LIN {X 0.039,Y -394.828,Z 1620.610,A 0.000,B 0.000,C 90.000,E1 109.812} C_DIS
LIN {X -0.087,Y -410.950,Z 1620.598,A 0.000,B 0.000,C 90.000,E1 107.583} C_DIS
LIN {X 0.069,Y -428.624,Z 1620.585,A 0.000,B 0.000,C 90.000,E1 105.371} C_DIS
LIN {X 0.081,Y -447.896,Z 1620.574,A 0.000,B 0.000,C 90.000,E1 103.244} C_DIS
LIN {X -0.189,Y -468.016,Z 1620.563,A 0.000,B 0.000,C 90.000,E1 101.299} C_DIS
LIN {X -0.227,Y -491.296,Z 1620.551,A 0.000,B 0.000,C 90.000,E1 99.265} C_DIS
LIN {X 0.069,Y -496.545,Z 1620.549,A 0.000,B 0.000,C 90.000,E1 98.803} C_DIS
LIN {X -0.222,Y -498.760,Z 1620.548,A 0.000,B 0.000,C 90.000,E1 98.624} C_DIS
LIN {X -0.096,Y -500.441,Z 1620.547,A 0.000,B 0.000,C 90.000,E1 98.398} C_DIS
LIN {X -0.170,Y -501.913,Z 1620.545,A 0.000,B 0.000,C 90.000,E1 98.163} C_DIS
LIN {X 0.252,Y -503.003,Z 1620.544,A 0.000,B 0.000,C 90.000,E1 97.871} C_DIS
LIN {X 0.048,Y -504.268,Z 1620.541,A 0.000,B 0.000,C 90.000,E1 97.409} C_DIS
LIN {X -0.150,Y -504.485,Z 1620.538,A 0.000,B 0.000,C 90.000,E1 96.947} C_DIS
LIN {X 0.160,Y -503.694,Z 1620.536,A 0.000,B 0.000,C 90.000,E1 96.429} C_DIS
LIN {X -0.030,Y -501.759,Z 1620.533,A 0.000,B 0.000,C 90.000,E1 95.967} C_DIS
LIN {X 0.225,Y -498.522,Z 1620.530,A 0.000,B 0.000,C 90.000,E1 95.454} C_DIS
LIN {X 0.209,Y -485.108,Z 1620.520,A 0.000,B 0.000,C 90.000,E1 93.498} C_DIS
LIN {X 0.202,Y -474.979,Z 1620.511,A 0.000,B 0.000,C 90.000,E1 92.007} C_DIS
LIN {X 0.024,Y -464.430,Z 1620.503,A 0.000,B 0.000,C 90.000,E1 90.516} C_DIS
LIN {X 0.121,Y -453.568,Z 1620.494,A 0.000,B 0.000,C 90.000,E1 88.969} C_DIS
LIN {X -0.158,Y -444.053,Z 1620.487,A 0.000,B 0.000,C 90.000,E1 87.707} C_DIS
LIN {X 0.033,Y -432.154,Z 1620.478,A 0.000,B 0.000,C 90.000,E1 86.102} C_DIS
LIN {X -0.096,Y -416.231,Z 1620.466,A 0.000,B 0.000,C 90.000,E1 83.970} C_DIS
LIN {X -0.079,Y -399.065,Z 1620.453,A 0.000,B 0.000,C 90.000,E1 81.489} C_DIS
LIN {X 0.091,Y -381.295,Z 1620.437,A 0.000,B 0.000,C 90.000,E1 78.634} C_DIS
LIN {X -0.092,Y -366.244,Z 1620.422,A 0.000,B 0.000,C 90.000,E1 76.047} C_DIS
LIN {X -0.121,Y -354.890,Z 1620.411,A 0.000,B 0.000,C 90.000,E1 73.976} C_DIS
LIN {X 0.056,Y -339.308,Z 1620.394,A 0.000,B 0.000,C 90.000,E1 70.913} C_DIS
LIN {X 0.117,Y -325.813,Z 1620.378,A 0.000,B 0.000,C 90.000,E1 68.103} C_DIS
LIN {X 0.153,Y -310.778,Z 1620.359,A 0.000,B 0.000,C 90.000,E1 64.588} C_DIS
LIN {X -0.117,Y -301.768,Z 1620.346,A 0.000,B 0.000,C 90.000,E1 62.359} C_DIS
LIN {X 0.106,Y -292.615,Z 1620.333,A 0.000,B 0.000,C 90.000,E1 59.999} C_DIS
LIN {X 0.041,Y -284.397,Z 1620.322,A 0.000,B 0.000,C 90.000,E1 57.995} C_DIS
LIN {X 0.019,Y -277.272,Z 1620.313,A 0.000,B 0.000,C 90.000,E1 56.294} C_DIS
LIN {X 0.123,Y -268.440,Z 1620.301,A 0.000,B 0.000,C 90.000,E1 54.196} C_DIS
LIN {X 0.060,Y -258.267,Z 1620.287,A 0.000,B 0.000,C 90.000,E1 51.743} C_DIS
LIN {X 0.110,Y -247.009,Z 1620.271,A 0.000,B 0.000,C 90.000,E1 48.852} C_DIS
LIN {X -0.019,Y -235.570,Z 1620.253,A 0.000,B 0.000,C 90.000,E1 45.567} C_DIS
LIN {X 0.043,Y -225.173,Z 1620.234,A 0.000,B 0.000,C 90.000,E1 42.162} C_DIS
LIN {X -0.046,Y -216.778,Z 1620.217,A 0.000,B 0.000,C 90.000,E1 39.116} C_DIS
LIN {X -0.102,Y -209.208,Z 1620.200,A 0.000,B 0.000,C 90.000,E1 36.011} C_DIS
LIN {X -0.074,Y -202.410,Z 1620.182,A 0.000,B 0.000,C 90.000,E1 32.832} C_DIS
LIN {X 0.013,Y -196.332,Z 1620.164,A 0.000,B 0.000,C 90.000,E1 29.589} C_DIS
LIN {X -0.096,Y -190.985,Z 1620.146,A 0.000,B 0.000,C 90.000,E1 26.360} C_DIS
LIN {X 0.019,Y -186.372,Z 1620.128,A 0.000,B 0.000,C 90.000,E1 23.025} C_DIS
LIN {X 0.023,Y -181.503,Z 1620.105,A 0.000,B 0.000,C 90.000,E1 18.852} C_DIS
LIN {X -0.016,Y -177.501,Z 1620.081,A 0.000,B 0.000,C 90.000,E1 14.647} C_DIS
LIN {X 0.063,Y -174.184,Z 1620.058,A 0.000,B 0.000,C 90.000,E1 10.366} C_DIS
LIN {X 0.061,Y -171.420,Z 1620.029,A 0.000,B 0.000,C 90.000,E1 5.220} C_DIS
LIN {X 0.000,Y -169.706,Z 1620.000,A 0.000,B 0.000,C 90.000,E1 360.000} C_DIS
LIN {X 0.005,Y -170.849,Z 1619.930,A 0.000,B 0.000,C 90.000,E1 347.409} C_DIS
LIN {X 0.018,Y -173.863,Z 1619.901,A 0.000,B 0.000,C 90.000,E1 342.236} C_DIS
LIN {X -0.034,Y -177.684,Z 1619.878,A 0.000,B 0.000,C 90.000,E1 337.975} C_DIS
LIN {X -0.054,Y -181.799,Z 1619.859,A 0.000,B 0.000,C 90.000,E1 334.588} C_DIS
LIN {X 0.104,Y -186.773,Z 1619.840,A 0.000,B 0.000,C 90.000,E1 331.179} C_DIS
LIN {X 0.076,Y -192.581,Z 1619.822,A 0.000,B 0.000,C 90.000,E1 327.867} C_DIS
LIN {X 0.010,Y -199.125,Z 1619.803,A 0.000,B 0.000,C 90.000,E1 324.609} C_DIS
LIN {X 0.022,Y -206.480,Z 1619.785,A 0.000,B 0.000,C 90.000,E1 321.376} C_DIS
LIN {X -0.028,Y -213.691,Z 1619.770,A 0.000,B 0.000,C 90.000,E1 318.609} C_DIS
LIN {X -0.020,Y -222.947,Z 1619.753,A 0.000,B 0.000,C 90.000,E1 315.486} C_DIS
LIN {X -0.099,Y -233.261,Z 1619.736,A 0.000,B 0.000,C 90.000,E1 312.447} C_DIS
LIN {X 0.021,Y -240.378,Z 1619.725,A 0.000,B 0.000,C 90.000,E1 310.539} C_DIS
LIN {X -0.047,Y -248.275,Z 1619.715,A 0.000,B 0.000,C 90.000,E1 308.705} C_DIS
LIN {X 0.038,Y -258.830,Z 1619.703,A 0.000,B 0.000,C 90.000,E1 306.503} C_DIS
LIN {X 0.074,Y -274.871,Z 1619.687,A 0.000,B 0.000,C 90.000,E1 303.658} C_DIS
LIN {X 0.052,Y -288.392,Z 1619.676,A 0.000,B 0.000,C 90.000,E1 301.592} C_DIS
LIN {X -0.139,Y -307.952,Z 1619.661,A 0.000,B 0.000,C 90.000,E1 298.949} C_DIS
LIN {X -0.148,Y -322.812,Z 1619.650,A 0.000,B 0.000,C 90.000,E1 297.001} C_DIS
LIN {X -0.137,Y -335.094,Z 1619.641,A 0.000,B 0.000,C 90.000,E1 295.412} C_DIS
LIN {X 0.086,Y -349.411,Z 1619.631,A 0.000,B 0.000,C 90.000,E1 293.515} C_DIS
LIN {X -0.020,Y -363.824,Z 1619.621,A 0.000,B 0.000,C 90.000,E1 291.716} C_DIS
LIN {X -0.061,Y -373.411,Z 1619.614,A 0.000,B 0.000,C 90.000,E1 290.536} C_DIS
LIN {X 0.121,Y -380.238,Z 1619.609,A 0.000,B 0.000,C 90.000,E1 289.631} C_DIS
LIN {X 0.023,Y -388.598,Z 1619.603,A 0.000,B 0.000,C 90.000,E1 288.489} C_DIS
LIN {X -0.017,Y -394.281,Z 1619.598,A 0.000,B 0.000,C 90.000,E1 287.638} C_DIS
LIN {X -0.182,Y -397.729,Z 1619.595,A 0.000,B 0.000,C 90.000,E1 287.094} C_DIS
LIN {X 0.129,Y -402.189,Z 1619.590,A 0.000,B 0.000,C 90.000,E1 286.205} C_DIS
LIN {X 0.097,Y -405.842,Z 1619.585,A 0.000,B 0.000,C 90.000,E1 285.371} C_DIS
LIN {X -0.002,Y -407.799,Z 1619.582,A 0.000,B 0.000,C 90.000,E1 284.828} C_DIS
LIN {X -0.201,Y -409.417,Z 1619.579,A 0.000,B 0.000,C 90.000,E1 284.300} C_DIS
LIN {X 0.013,Y -410.583,Z 1619.576,A 0.000,B 0.000,C 90.000,E1 283.716} C_DIS
LIN {X -0.066,Y -411.312,Z 1619.573,A 0.000,B 0.000,C 90.000,E1 283.175} C_DIS
LIN {X 0.166,Y -411.580,Z 1619.570,A 0.000,B 0.000,C 90.000,E1 282.591} C_DIS
LIN {X 0.003,Y -411.346,Z 1619.567,A 0.000,B 0.000,C 90.000,E1 282.063} C_DIS
LIN {X -0.160,Y -410.620,Z 1619.564,A 0.000,B 0.000,C 90.000,E1 281.535} C_DIS
LIN {X 0.078,Y -409.270,Z 1619.561,A 0.000,B 0.000,C 90.000,E1 280.950} C_DIS
LIN {X -0.092,Y -407.390,Z 1619.558,A 0.000,B 0.000,C 90.000,E1 280.423} C_DIS
LIN {X 0.059,Y -404.789,Z 1619.555,A 0.000,B 0.000,C 90.000,E1 279.849} C_DIS
LIN {X -0.136,Y -401.553,Z 1619.552,A 0.000,B 0.000,C 90.000,E1 279.321} C_DIS
LIN {X -0.015,Y -397.674,Z 1619.549,A 0.000,B 0.000,C 90.000,E1 278.746} C_DIS
LIN {X 0.142,Y -393.240,Z 1619.545,A 0.000,B 0.000,C 90.000,E1 278.163} C_DIS
LIN {X -0.091,Y -385.513,Z 1619.541,A 0.000,B 0.000,C 90.000,E1 277.352} C_DIS
LIN {X 0.125,Y -379.865,Z 1619.538,A 0.000,B 0.000,C 90.000,E1 276.777} C_DIS
LIN {X -0.178,Y -373.999,Z 1619.535,A 0.000,B 0.000,C 90.000,E1 276.315} C_DIS
LIN {X 0.136,Y -367.955,Z 1619.532,A 0.000,B 0.000,C 90.000,E1 275.796} C_DIS
LIN {X -0.047,Y -361.745,Z 1619.530,A 0.000,B 0.000,C 90.000,E1 275.391} C_DIS
LIN {X -0.146,Y -352.071,Z 1619.527,A 0.000,B 0.000,C 90.000,E1 274.816} C_DIS
LIN {X -0.156,Y -342.525,Z 1619.524,A 0.000,B 0.000,C 90.000,E1 274.302} C_DIS
LIN {X 0.156,Y -332.645,Z 1619.521,A 0.000,B 0.000,C 90.000,E1 273.784} C_DIS
LIN {X 0.109,Y -323.028,Z 1619.519,A 0.000,B 0.000,C 90.000,E1 273.383} C_DIS
LIN {X -0.026,Y -313.116,Z 1619.517,A 0.000,B 0.000,C 90.000,E1 273.037} C_DIS
LIN {X -0.012,Y -306.390,Z 1619.516,A 0.000,B 0.000,C 90.000,E1 272.808} C_DIS
LIN {X -0.058,Y -295.571,Z 1619.514,A 0.000,B 0.000,C 90.000,E1 272.522} C_DIS
LIN {X -0.014,Y -287.863,Z 1619.513,A 0.000,B 0.000,C 90.000,E1 272.350} C_DIS
LIN {X -0.122,Y -279.479,Z 1619.512,A 0.000,B 0.000,C 90.000,E1 272.236} C_DIS
LIN {X -0.049,Y -258.995,Z 1619.511,A 0.000,B 0.000,C 90.000,E1 272.007} C_DIS
LIN {X 0.051,Y -231.617,Z 1619.510,A 0.000,B 0.000,C 90.000,E1 271.776} C_DIS
LIN {X 0.051,Y -219.103,Z 1619.510,A 0.000,B 0.000,C 90.000,E1 271.718} C_DIS
LIN {X 0.007,Y -211.613,Z 1619.510,A 0.000,B 0.000,C 90.000,E1 271.718} C_DIS
LIN {X -0.030,Y -181.312,Z 1619.510,A 0.000,B 0.000,C 90.000,E1 271.718} C_DIS
LIN {X -0.030,Y -181.559,Z 1619.500,A 0.000,B 0.000,C 90.000,E1 270.000} C_DIS
LIN {X -0.044,Y -180.847,Z 1619.472,A 0.000,B 0.000,C 90.000,E1 264.951} C_DIS
LIN {X 0.039,Y -178.956,Z 1619.444,A 0.000,B 0.000,C 90.000,E1 259.859} C_DIS
LIN {X -0.069,Y -177.357,Z 1619.430,A 0.000,B 0.000,C 90.000,E1 257.353} C_DIS
LIN {X 0.027,Y -175.528,Z 1619.411,A 0.000,B 0.000,C 90.000,E1 253.921} C_DIS
LIN {X 0.028,Y -172.264,Z 1619.387,A 0.000,B 0.000,C 90.000,E1 249.645} C_DIS
LIN {X 0.067,Y -171.743,Z 1619.382,A 0.000,B 0.000,C 90.000,E1 248.773} C_DIS
LIN {X -0.075,Y -167.341,Z 1619.353,A 0.000,B 0.000,C 90.000,E1 243.640} C_DIS
LIN {X 0.007,Y -166.727,Z 1619.349,A 0.000,B 0.000,C 90.000,E1 242.743} C_DIS
LIN {X -0.080,Y -162.707,Z 1619.324,A 0.000,B 0.000,C 90.000,E1 238.408} C_DIS
LIN {X -0.018,Y -161.397,Z 1619.315,A 0.000,B 0.000,C 90.000,E1 236.628} C_DIS
LIN {X 0.024,Y -157.390,Z 1619.290,A 0.000,B 0.000,C 90.000,E1 232.190} C_DIS
LIN {X -0.043,Y -155.386,Z 1619.275,A 0.000,B 0.000,C 90.000,E1 229.542} C_DIS
LIN {X -0.003,Y -151.722,Z 1619.250,A 0.000,B 0.000,C 90.000,E1 225.040} C_DIS
LIN {X 0.013,Y -149.915,Z 1619.235,A 0.000,B 0.000,C 90.000,E1 222.324} C_DIS
LIN {X -0.069,Y -146.770,Z 1619.210,A 0.000,B 0.000,C 90.000,E1 217.810} C_DIS
LIN {X 0.034,Y -145.339,Z 1619.195,A 0.000,B 0.000,C 90.000,E1 215.025} C_DIS
LIN {X -0.050,Y -142.417,Z 1619.164,A 0.000,B 0.000,C 90.000,E1 209.539} C_DIS
LIN {X 0.000,Y -141.403,Z 1619.149,A 0.000,B 0.000,C 90.000,E1 206.744} C_DIS
LIN {X -0.013,Y -139.356,Z 1619.112,A 0.000,B 0.000,C 90.000,E1 200.248} C_DIS
LIN {X -0.025,Y -138.797,Z 1619.097,A 0.000,B 0.000,C 90.000,E1 197.457} C_DIS
LIN {X 0.030,Y -138.348,Z 1619.055,A 0.000,B 0.000,C 90.000,E1 189.962} C_DIS
LIN {X 0.047,Y -139.373,Z 1619.009,A 0.000,B 0.000,C 90.000,E1 181.547} C_DIS
LIN {X -0.039,Y -141.262,Z 1618.973,A 0.000,B 0.000,C 90.000,E1 175.065} C_DIS
LIN {X 0.060,Y -142.629,Z 1618.957,A 0.000,B 0.000,C 90.000,E1 172.243} C_DIS
LIN {X 0.011,Y -144.955,Z 1618.931,A 0.000,B 0.000,C 90.000,E1 167.645} C_DIS
LIN {X 0.003,Y -147.582,Z 1618.911,A 0.000,B 0.000,C 90.000,E1 163.976} C_DIS
LIN {X 0.033,Y -150.196,Z 1618.891,A 0.000,B 0.000,C 90.000,E1 160.315} C_DIS
LIN {X -0.040,Y -153.578,Z 1618.871,A 0.000,B 0.000,C 90.000,E1 156.719} C_DIS
LIN {X -0.050,Y -156.994,Z 1618.851,A 0.000,B 0.000,C 90.000,E1 153.127} C_DIS
LIN {X 0.023,Y -161.109,Z 1618.831,A 0.000,B 0.000,C 90.000,E1 149.537} C_DIS
LIN {X -0.032,Y -163.212,Z 1618.821,A 0.000,B 0.000,C 90.000,E1 147.788} C_DIS
LIN {X -0.028,Y -167.641,Z 1618.802,A 0.000,B 0.000,C 90.000,E1 144.276} C_DIS
LIN {X -0.013,Y -171.466,Z 1618.787,A 0.000,B 0.000,C 90.000,E1 141.662} C_DIS
LIN {X -0.082,Y -176.392,Z 1618.768,A 0.000,B 0.000,C 90.000,E1 138.243} C_DIS
LIN {X 0.039,Y -180.686,Z 1618.754,A 0.000,B 0.000,C 90.000,E1 135.648} C_DIS
LIN {X 0.021,Y -186.089,Z 1618.735,A 0.000,B 0.000,C 90.000,E1 132.285} C_DIS
LIN {X -0.043,Y -190.726,Z 1618.721,A 0.000,B 0.000,C 90.000,E1 129.806} C_DIS
LIN {X -0.011,Y -196.478,Z 1618.703,A 0.000,B 0.000,C 90.000,E1 126.503} C_DIS
LIN {X -0.044,Y -201.259,Z 1618.689,A 0.000,B 0.000,C 90.000,E1 124.072} C_DIS
LIN {X 0.113,Y -205.676,Z 1618.676,A 0.000,B 0.000,C 90.000,E1 121.592} C_DIS
LIN {X 0.144,Y -324.533,Z 1618.676,A 0.000,B 0.000,C 90.000,E1 121.592} C_DIS
LIN {X -0.063,Y -326.700,Z 1618.675,A 0.000,B 0.000,C 90.000,E1 121.592} C_DIS
LIN {X 0.062,Y -330.806,Z 1618.674,A 0.000,B 0.000,C 90.000,E1 121.386} C_DIS
LIN {X 0.015,Y -333.192,Z 1618.673,A 0.000,B 0.000,C 90.000,E1 121.209} C_DIS
LIN {X -0.019,Y -336.461,Z 1618.671,A 0.000,B 0.000,C 90.000,E1 120.846} C_DIS
LIN {X -0.002,Y -338.376,Z 1618.670,A 0.000,B 0.000,C 90.000,E1 120.541} C_DIS
LIN {X -0.103,Y -339.868,Z 1618.668,A 0.000,B 0.000,C 90.000,E1 120.256} C_DIS
LIN {X 0.087,Y -351.799,Z 1618.653,A 0.000,B 0.000,C 90.000,E1 117.462} C_DIS
LIN {X -0.014,Y -365.163,Z 1618.638,A 0.000,B 0.000,C 90.000,E1 114.771} C_DIS
LIN {X -0.202,Y -380.085,Z 1618.623,A 0.000,B 0.000,C 90.000,E1 112.153} C_DIS
LIN {X 0.074,Y -394.768,Z 1618.610,A 0.000,B 0.000,C 90.000,E1 109.812} C_DIS
LIN {X -0.052,Y -410.887,Z 1618.598,A 0.000,B 0.000,C 90.000,E1 107.583} C_DIS
LIN {X 0.104,Y -428.557,Z 1618.585,A 0.000,B 0.000,C 90.000,E1 105.371} C_DIS
LIN {X 0.115,Y -447.826,Z 1618.574,A 0.000,B 0.000,C 90.000,E1 103.244} C_DIS
LIN {X -0.158,Y -467.946,Z 1618.563,A 0.000,B 0.000,C 90.000,E1 101.299} C_DIS
LIN {X -0.197,Y -491.224,Z 1618.551,A 0.000,B 0.000,C 90.000,E1 99.265} C_DIS
LIN {X 0.098,Y -496.470,Z 1618.549,A 0.000,B 0.000,C 90.000,E1 98.803} C_DIS
LIN {X -0.195,Y -498.664,Z 1618.548,A 0.000,B 0.000,C 90.000,E1 98.624} C_DIS
LIN {X -0.070,Y -500.332,Z 1618.547,A 0.000,B 0.000,C 90.000,E1 98.398} C_DIS
LIN {X -0.144,Y -501.791,Z 1618.545,A 0.000,B 0.000,C 90.000,E1 98.163} C_DIS
LIN {X 0.277,Y -502.872,Z 1618.544,A 0.000,B 0.000,C 90.000,E1 97.871} C_DIS
LIN {X 0.073,Y -504.121,Z 1618.541,A 0.000,B 0.000,C 90.000,E1 97.409} C_DIS
LIN {X -0.126,Y -504.326,Z 1618.539,A 0.000,B 0.000,C 90.000,E1 96.947} C_DIS
LIN {X 0.182,Y -503.521,Z 1618.536,A 0.000,B 0.000,C 90.000,E1 96.429} C_DIS
LIN {X -0.008,Y -501.569,Z 1618.533,A 0.000,B 0.000,C 90.000,E1 95.967} C_DIS
LIN {X -0.251,Y -498.321,Z 1618.530,A 0.000,B 0.000,C 90.000,E1 95.511} C_DIS
LIN {X 0.225,Y -484.929,Z 1618.520,A 0.000,B 0.000,C 90.000,E1 93.498} C_DIS
LIN {X -0.089,Y -476.522,Z 1618.513,A 0.000,B 0.000,C 90.000,E1 92.293} C_DIS
LIN {X -0.039,Y -467.833,Z 1618.506,A 0.000,B 0.000,C 90.000,E1 91.031} C_DIS
LIN {X 0.117,Y -457.058,Z 1618.497,A 0.000,B 0.000,C 90.000,E1 89.484} C_DIS
LIN {X -0.127,Y -447.716,Z 1618.490,A 0.000,B 0.000,C 90.000,E1 88.224} C_DIS
LIN {X -0.041,Y -437.969,Z 1618.483,A 0.000,B 0.000,C 90.000,E1 86.906} C_DIS
LIN {X -0.201,Y -423.966,Z 1618.472,A 0.000,B 0.000,C 90.000,E1 85.065} C_DIS
LIN {X 0.076,Y -404.437,Z 1618.457,A 0.000,B 0.000,C 90.000,E1 82.299} C_DIS
LIN {X -0.003,Y -384.581,Z 1618.440,A 0.000,B 0.000,C 90.000,E1 79.218} C_DIS
LIN {X -0.183,Y -367.707,Z 1618.424,A 0.000,B 0.000,C 90.000,E1 76.353} C_DIS
LIN {X -0.095,Y -356.322,Z 1618.412,A 0.000,B 0.000,C 90.000,E1 74.267} C_DIS
LIN {X 0.125,Y -342.171,Z 1618.397,A 0.000,B 0.000,C 90.000,E1 71.511} C_DIS
LIN {X -0.114,Y -331.562,Z 1618.385,A 0.000,B 0.000,C 90.000,E1 69.390} C_DIS
LIN {X -0.012,Y -318.580,Z 1618.370,A 0.000,B 0.000,C 90.000,E1 66.538} C_DIS
LIN {X 0.027,Y -305.465,Z 1618.352,A 0.000,B 0.000,C 90.000,E1 63.307} C_DIS
LIN {X 0.178,Y -297.715,Z 1618.341,A 0.000,B 0.000,C 90.000,E1 61.307} C_DIS
LIN {X 0.062,Y -289.753,Z 1618.330,A 0.000,B 0.000,C 90.000,E1 59.331} C_DIS
LIN {X -0.055,Y -281.414,Z 1618.318,A 0.000,B 0.000,C 90.000,E1 57.327} C_DIS
LIN {X -0.026,Y -272.670,Z 1618.307,A 0.000,B 0.000,C 90.000,E1 55.261} C_DIS
LIN {X -0.097,Y -260.924,Z 1618.291,A 0.000,B 0.000,C 90.000,E1 52.477} C_DIS
LIN {X 0.043,Y -248.085,Z 1618.273,A 0.000,B 0.000,C 90.000,E1 49.218} C_DIS
LIN {X 0.124,Y -236.548,Z 1618.255,A 0.000,B 0.000,C 90.000,E1 45.891} C_DIS
LIN {X -0.061,Y -227.183,Z 1618.238,A 0.000,B 0.000,C 90.000,E1 42.933} C_DIS
LIN {X 0.045,Y -218.658,Z 1618.221,A 0.000,B 0.000,C 90.000,E1 39.850} C_DIS
LIN {X 0.032,Y -210.909,Z 1618.204,A 0.000,B 0.000,C 90.000,E1 36.744} C_DIS
LIN {X 0.047,Y -203.960,Z 1618.187,A 0.000,B 0.000,C 90.000,E1 33.579} C_DIS
LIN {X 0.001,Y -197.736,Z 1618.169,A 0.000,B 0.000,C 90.000,E1 30.384} C_DIS
LIN {X 0.015,Y -192.226,Z 1618.151,A 0.000,B 0.000,C 90.000,E1 27.129} C_DIS
LIN {X 0.064,Y -187.465,Z 1618.132,A 0.000,B 0.000,C 90.000,E1 23.823} C_DIS
LIN {X -0.014,Y -182.446,Z 1618.109,A 0.000,B 0.000,C 90.000,E1 19.685} C_DIS
LIN {X -0.027,Y -178.324,Z 1618.086,A 0.000,B 0.000,C 90.000,E1 15.481} C_DIS
LIN {X -0.054,Y -174.857,Z 1618.062,A 0.000,B 0.000,C 90.000,E1 11.243} C_DIS
LIN {X -0.001,Y -171.922,Z 1618.034,A 0.000,B 0.000,C 90.000,E1 6.087} C_DIS
LIN {X -0.002,Y -170.095,Z 1618.005,A 0.000,B 0.000,C 90.000,E1 0.917} C_DIS
LIN {X 0.019,Y -171.031,Z 1617.930,A 0.000,B 0.000,C 90.000,E1 347.409} C_DIS
LIN {X 0.040,Y -174.049,Z 1617.901,A 0.000,B 0.000,C 90.000,E1 342.236} C_DIS
LIN {X -0.006,Y -177.888,Z 1617.878,A 0.000,B 0.000,C 90.000,E1 337.975} C_DIS
LIN {X -0.021,Y -181.997,Z 1617.859,A 0.000,B 0.000,C 90.000,E1 334.588} C_DIS
LIN {X -0.110,Y -186.951,Z 1617.840,A 0.000,B 0.000,C 90.000,E1 331.257} C_DIS
LIN {X -0.043,Y -192.755,Z 1617.822,A 0.000,B 0.000,C 90.000,E1 327.916} C_DIS
LIN {X 0.061,Y -199.275,Z 1617.803,A 0.000,B 0.000,C 90.000,E1 324.609} C_DIS
LIN {X 0.078,Y -206.626,Z 1617.786,A 0.000,B 0.000,C 90.000,E1 321.376} C_DIS
LIN {X 0.034,Y -213.812,Z 1617.770,A 0.000,B 0.000,C 90.000,E1 318.609} C_DIS
LIN {X 0.048,Y -223.026,Z 1617.753,A 0.000,B 0.000,C 90.000,E1 315.486} C_DIS
LIN {X -0.027,Y -233.270,Z 1617.736,A 0.000,B 0.000,C 90.000,E1 312.447} C_DIS
LIN {X 0.095,Y -240.362,Z 1617.725,A 0.000,B 0.000,C 90.000,E1 310.539} C_DIS
LIN {X 0.030,Y -248.226,Z 1617.715,A 0.000,B 0.000,C 90.000,E1 308.705} C_DIS
LIN {X 0.086,Y -256.901,Z 1617.705,A 0.000,B 0.000,C 90.000,E1 306.870} C_DIS
LIN {X -0.062,Y -270.581,Z 1617.691,A 0.000,B 0.000,C 90.000,E1 304.405} C_DIS
LIN {X 0.066,Y -283.648,Z 1617.679,A 0.000,B 0.000,C 90.000,E1 302.291} C_DIS
LIN {X -0.078,Y -305.338,Z 1617.663,A 0.000,B 0.000,C 90.000,E1 299.283} C_DIS
LIN {X 0.015,Y -320.212,Z 1617.652,A 0.000,B 0.000,C 90.000,E1 297.308} C_DIS
LIN {X -0.006,Y -332.518,Z 1617.643,A 0.000,B 0.000,C 90.000,E1 295.720} C_DIS
LIN {X 0.023,Y -344.539,Z 1617.634,A 0.000,B 0.000,C 90.000,E1 294.155} C_DIS
LIN {X -0.033,Y -358.906,Z 1617.624,A 0.000,B 0.000,C 90.000,E1 292.333} C_DIS
LIN {X -0.022,Y -371.000,Z 1617.616,A 0.000,B 0.000,C 90.000,E1 290.844} C_DIS
LIN {X -0.112,Y -380.176,Z 1617.609,A 0.000,B 0.000,C 90.000,E1 289.685} C_DIS
LIN {X 0.150,Y -388.558,Z 1617.603,A 0.000,B 0.000,C 90.000,E1 288.489} C_DIS
LIN {X -0.045,Y -392.474,Z 1617.600,A 0.000,B 0.000,C 90.000,E1 287.946} C_DIS
LIN {X -0.052,Y -397.730,Z 1617.595,A 0.000,B 0.000,C 90.000,E1 287.094} C_DIS
LIN {X 0.186,Y -400.872,Z 1617.592,A 0.000,B 0.000,C 90.000,E1 286.496} C_DIS
LIN {X 0.144,Y -404.846,Z 1617.587,A 0.000,B 0.000,C 90.000,E1 285.662} C_DIS
LIN {X 0.132,Y -407.961,Z 1617.583,A 0.000,B 0.000,C 90.000,E1 284.828} C_DIS
LIN {X -0.065,Y -409.606,Z 1617.579,A 0.000,B 0.000,C 90.000,E1 284.300} C_DIS
LIN {X 0.150,Y -410.830,Z 1617.576,A 0.000,B 0.000,C 90.000,E1 283.716} C_DIS
LIN {X 0.072,Y -411.528,Z 1617.573,A 0.000,B 0.000,C 90.000,E1 283.175} C_DIS
LIN {X -0.096,Y -411.871,Z 1617.570,A 0.000,B 0.000,C 90.000,E1 282.647} C_DIS
LIN {X 0.143,Y -411.669,Z 1617.567,A 0.000,B 0.000,C 90.000,E1 282.063} C_DIS
LIN {X -0.018,Y -410.975,Z 1617.564,A 0.000,B 0.000,C 90.000,E1 281.535} C_DIS
LIN {X 0.222,Y -409.715,Z 1617.561,A 0.000,B 0.000,C 90.000,E1 280.950} C_DIS
LIN {X -0.021,Y -407.846,Z 1617.558,A 0.000,B 0.000,C 90.000,E1 280.433} C_DIS
LIN {X -0.193,Y -405.326,Z 1617.555,A 0.000,B 0.000,C 90.000,E1 279.905} C_DIS
LIN {X 0.013,Y -402.111,Z 1617.552,A 0.000,B 0.000,C 90.000,E1 279.321} C_DIS
LIN {X 0.136,Y -398.316,Z 1617.549,A 0.000,B 0.000,C 90.000,E1 278.746} C_DIS
LIN {X -0.095,Y -393.879,Z 1617.546,A 0.000,B 0.000,C 90.000,E1 278.219} C_DIS
LIN {X -0.017,Y -388.853,Z 1617.542,A 0.000,B 0.000,C 90.000,E1 277.644} C_DIS
LIN {X 0.080,Y -383.328,Z 1617.539,A 0.000,B 0.000,C 90.000,E1 277.068} C_DIS
LIN {X -0.047,Y -374.634,Z 1617.535,A 0.000,B 0.000,C 90.000,E1 276.315} C_DIS
LIN {X -0.094,Y -368.553,Z 1617.532,A 0.000,B 0.000,C 90.000,E1 275.853} C_DIS
LIN {X 0.085,Y -362.325,Z 1617.530,A 0.000,B 0.000,C 90.000,E1 275.391} C_DIS
LIN {X -0.053,Y -352.665,Z 1617.527,A 0.000,B 0.000,C 90.000,E1 274.821} C_DIS
LIN {X -0.041,Y -343.024,Z 1617.524,A 0.000,B 0.000,C 90.000,E1 274.302} C_DIS
LIN {X 0.159,Y -336.597,Z 1617.522,A 0.000,B 0.000,C 90.000,E1 273.955} C_DIS
LIN {X 0.021,Y -326.896,Z 1617.520,A 0.000,B 0.000,C 90.000,E1 273.555} C_DIS
LIN {X 0.112,Y -317.012,Z 1617.518,A 0.000,B 0.000,C 90.000,E1 273.154} C_DIS
LIN {X 0.111,Y -306.941,Z 1617.516,A 0.000,B 0.000,C 90.000,E1 272.808} C_DIS
LIN {X 0.049,Y -296.202,Z 1617.514,A 0.000,B 0.000,C 90.000,E1 272.522} C_DIS
LIN {X 0.083,Y -288.602,Z 1617.513,A 0.000,B 0.000,C 90.000,E1 272.350} C_DIS
LIN {X -0.026,Y -280.515,Z 1617.512,A 0.000,B 0.000,C 90.000,E1 272.236} C_DIS
LIN {X 0.058,Y -261.144,Z 1617.511,A 0.000,B 0.000,C 90.000,E1 272.007} C_DIS
LIN {X -0.096,Y -234.493,Z 1617.510,A 0.000,B 0.000,C 90.000,E1 271.833} C_DIS
LIN {X 0.094,Y -219.614,Z 1617.510,A 0.000,B 0.000,C 90.000,E1 271.718} C_DIS
LIN {X 0.042,Y -181.308,Z 1617.510,A 0.000,B 0.000,C 90.000,E1 271.718} C_DIS
LIN {X 0.046,Y -181.563,Z 1617.500,A 0.000,B 0.000,C 90.000,E1 270.000} C_DIS
LIN {X 0.032,Y -180.853,Z 1617.472,A 0.000,B 0.000,C 90.000,E1 264.951} C_DIS
LIN {X -0.063,Y -178.964,Z 1617.444,A 0.000,B 0.000,C 90.000,E1 259.916} C_DIS
LIN {X 0.005,Y -177.372,Z 1617.430,A 0.000,B 0.000,C 90.000,E1 257.353} C_DIS
LIN {X -0.068,Y -175.548,Z 1617.411,A 0.000,B 0.000,C 90.000,E1 253.976} C_DIS
LIN {X -0.059,Y -172.279,Z 1617.387,A 0.000,B 0.000,C 90.000,E1 249.699} C_DIS
LIN {X -0.020,Y -171.758,Z 1617.382,A 0.000,B 0.000,C 90.000,E1 248.827} C_DIS
LIN {X -0.003,Y -167.358,Z 1617.354,A 0.000,B 0.000,C 90.000,E1 243.640} C_DIS
LIN {X 0.079,Y -166.747,Z 1617.349,A 0.000,B 0.000,C 90.000,E1 242.743} C_DIS
LIN {X -0.009,Y -162.727,Z 1617.324,A 0.000,B 0.000,C 90.000,E1 238.408} C_DIS
LIN {X 0.052,Y -161.417,Z 1617.315,A 0.000,B 0.000,C 90.000,E1 236.628} C_DIS
LIN {X 0.093,Y -157.410,Z 1617.290,A 0.000,B 0.000,C 90.000,E1 232.190} C_DIS
LIN {X 0.025,Y -155.411,Z 1617.275,A 0.000,B 0.000,C 90.000,E1 229.542} C_DIS
LIN {X -0.043,Y -151.739,Z 1617.250,A 0.000,B 0.000,C 90.000,E1 225.081} C_DIS
LIN {X -0.031,Y -149.936,Z 1617.235,A 0.000,B 0.000,C 90.000,E1 222.366} C_DIS
LIN {X -0.003,Y -146.784,Z 1617.210,A 0.000,B 0.000,C 90.000,E1 217.810} C_DIS
LIN {X 0.100,Y -145.357,Z 1617.195,A 0.000,B 0.000,C 90.000,E1 215.025} C_DIS
LIN {X 0.015,Y -142.427,Z 1617.164,A 0.000,B 0.000,C 90.000,E1 209.539} C_DIS
LIN {X 0.064,Y -141.415,Z 1617.149,A 0.000,B 0.000,C 90.000,E1 206.744} C_DIS
LIN {X 0.051,Y -139.360,Z 1617.113,A 0.000,B 0.000,C 90.000,E1 200.248} C_DIS
LIN {X 0.039,Y -138.803,Z 1617.097,A 0.000,B 0.000,C 90.000,E1 197.457} C_DIS
LIN {X -0.042,Y -138.349,Z 1617.056,A 0.000,B 0.000,C 90.000,E1 190.018} C_DIS
LIN {X -0.028,Y -139.365,Z 1617.009,A 0.000,B 0.000,C 90.000,E1 181.604} C_DIS
LIN {X 0.025,Y -141.250,Z 1616.973,A 0.000,B 0.000,C 90.000,E1 175.065} C_DIS
LIN {X -0.017,Y -142.619,Z 1616.957,A 0.000,B 0.000,C 90.000,E1 172.299} C_DIS
LIN {X -0.064,Y -144.938,Z 1616.932,A 0.000,B 0.000,C 90.000,E1 167.701} C_DIS
LIN {X 0.069,Y -147.566,Z 1616.911,A 0.000,B 0.000,C 90.000,E1 163.976} C_DIS
LIN {X -0.041,Y -150.174,Z 1616.891,A 0.000,B 0.000,C 90.000,E1 160.369} C_DIS
LIN {X -0.033,Y -153.551,Z 1616.871,A 0.000,B 0.000,C 90.000,E1 156.741} C_DIS
LIN {X 0.020,Y -156.968,Z 1616.851,A 0.000,B 0.000,C 90.000,E1 153.127} C_DIS
LIN {X -0.046,Y -161.077,Z 1616.831,A 0.000,B 0.000,C 90.000,E1 149.587} C_DIS
LIN {X 0.039,Y -163.183,Z 1616.821,A 0.000,B 0.000,C 90.000,E1 147.788} C_DIS
LIN {X 0.045,Y -167.606,Z 1616.802,A 0.000,B 0.000,C 90.000,E1 144.276} C_DIS
LIN {X -0.046,Y -171.434,Z 1616.787,A 0.000,B 0.000,C 90.000,E1 141.698} C_DIS
LIN {X -0.008,Y -176.354,Z 1616.768,A 0.000,B 0.000,C 90.000,E1 138.243} C_DIS
LIN {X -0.011,Y -180.645,Z 1616.754,A 0.000,B 0.000,C 90.000,E1 135.688} C_DIS
LIN {X -0.027,Y -186.047,Z 1616.735,A 0.000,B 0.000,C 90.000,E1 132.324} C_DIS
LIN {X 0.036,Y -190.683,Z 1616.721,A 0.000,B 0.000,C 90.000,E1 129.806} C_DIS
LIN {X 0.069,Y -196.435,Z 1616.703,A 0.000,B 0.000,C 90.000,E1 126.503} C_DIS
LIN {X 0.035,Y -201.219,Z 1616.689,A 0.000,B 0.000,C 90.000,E1 124.072} C_DIS
LIN {X -0.021,Y -205.597,Z 1616.676,A 0.000,B 0.000,C 90.000,E1 121.671} C_DIS
LIN {X -0.068,Y -323.917,Z 1616.676,A 0.000,B 0.000,C 90.000,E1 121.671} C_DIS
LIN {X 0.067,Y -327.100,Z 1616.676,A 0.000,B 0.000,C 90.000,E1 121.592} C_DIS
LIN {X 0.020,Y -330.883,Z 1616.675,A 0.000,B 0.000,C 90.000,E1 121.416} C_DIS
LIN {X -0.138,Y -333.198,Z 1616.674,A 0.000,B 0.000,C 90.000,E1 121.258} C_DIS
LIN {X -0.060,Y -336.403,Z 1616.672,A 0.000,B 0.000,C 90.000,E1 120.875} C_DIS
LIN {X 0.107,Y -338.311,Z 1616.670,A 0.000,B 0.000,C 90.000,E1 120.541} C_DIS
LIN {X 0.128,Y -341.061,Z 1616.666,A 0.000,B 0.000,C 90.000,E1 119.922} C_DIS
LIN {X 0.041,Y -353.125,Z 1616.651,A 0.000,B 0.000,C 90.000,E1 117.180} C_DIS
LIN {X 0.146,Y -366.644,Z 1616.636,A 0.000,B 0.000,C 90.000,E1 114.463} C_DIS
LIN {X -0.114,Y -379.982,Z 1616.623,A 0.000,B 0.000,C 90.000,E1 112.153} C_DIS
LIN {X 0.162,Y -394.656,Z 1616.610,A 0.000,B 0.000,C 90.000,E1 109.812} C_DIS
LIN {X 0.038,Y -410.767,Z 1616.598,A 0.000,B 0.000,C 90.000,E1 107.583} C_DIS
LIN {X 0.194,Y -428.427,Z 1616.586,A 0.000,B 0.000,C 90.000,E1 105.371} C_DIS
LIN {X -0.232,Y -447.688,Z 1616.574,A 0.000,B 0.000,C 90.000,E1 103.300} C_DIS
LIN {X -0.074,Y -467.805,Z 1616.563,A 0.000,B 0.000,C 90.000,E1 101.299} C_DIS
LIN {X -0.118,Y -491.081,Z 1616.551,A 0.000,B 0.000,C 90.000,E1 99.265} C_DIS
LIN {X 0.176,Y -496.326,Z 1616.549,A 0.000,B 0.000,C 90.000,E1 98.803} C_DIS
LIN {X -0.117,Y -498.517,Z 1616.548,A 0.000,B 0.000,C 90.000,E1 98.624} C_DIS
LIN {X 0.007,Y -500.183,Z 1616.547,A 0.000,B 0.000,C 90.000,E1 98.398} C_DIS
LIN {X -0.068,Y -501.639,Z 1616.545,A 0.000,B 0.000,C 90.000,E1 98.163} C_DIS
LIN {X -0.214,Y -502.719,Z 1616.544,A 0.000,B 0.000,C 90.000,E1 97.936} C_DIS
LIN {X 0.148,Y -503.963,Z 1616.541,A 0.000,B 0.000,C 90.000,E1 97.409} C_DIS
LIN {X -0.051,Y -504.166,Z 1616.539,A 0.000,B 0.000,C 90.000,E1 96.947} C_DIS
LIN {X 0.256,Y -503.358,Z 1616.536,A 0.000,B 0.000,C 90.000,E1 96.429} C_DIS
LIN {X 0.064,Y -501.402,Z 1616.533,A 0.000,B 0.000,C 90.000,E1 95.967} C_DIS
LIN {X -0.179,Y -498.159,Z 1616.531,A 0.000,B 0.000,C 90.000,E1 95.511} C_DIS
LIN {X -0.193,Y -484.797,Z 1616.520,A 0.000,B 0.000,C 90.000,E1 93.555} C_DIS
LIN {X -0.198,Y -474.705,Z 1616.511,A 0.000,B 0.000,C 90.000,E1 92.064} C_DIS
LIN {X 0.093,Y -464.168,Z 1616.503,A 0.000,B 0.000,C 90.000,E1 90.516} C_DIS
LIN {X 0.182,Y -453.245,Z 1616.494,A 0.000,B 0.000,C 90.000,E1 88.969} C_DIS
LIN {X -0.102,Y -443.761,Z 1616.487,A 0.000,B 0.000,C 90.000,E1 87.707} C_DIS
LIN {X -0.068,Y -433.847,Z 1616.480,A 0.000,B 0.000,C 90.000,E1 86.388} C_DIS
LIN {X 0.117,Y -419.840,Z 1616.469,A 0.000,B 0.000,C 90.000,E1 84.489} C_DIS
LIN {X -0.048,Y -398.743,Z 1616.453,A 0.000,B 0.000,C 90.000,E1 81.489} C_DIS
LIN {X 0.110,Y -380.986,Z 1616.437,A 0.000,B 0.000,C 90.000,E1 78.634} C_DIS
LIN {X -0.080,Y -365.939,Z 1616.422,A 0.000,B 0.000,C 90.000,E1 76.047} C_DIS
LIN {X -0.116,Y -354.567,Z 1616.411,A 0.000,B 0.000,C 90.000,E1 73.976} C_DIS
LIN {X 0.036,Y -342.026,Z 1616.397,A 0.000,B 0.000,C 90.000,E1 71.529} C_DIS
LIN {X -0.097,Y -331.433,Z 1616.385,A 0.000,B 0.000,C 90.000,E1 69.390} C_DIS
LIN {X 0.000,Y -318.421,Z 1616.370,A 0.000,B 0.000,C 90.000,E1 66.538} C_DIS
LIN {X 0.035,Y -305.313,Z 1616.352,A 0.000,B 0.000,C 90.000,E1 63.307} C_DIS
LIN {X 0.040,Y -297.594,Z 1616.341,A 0.000,B 0.000,C 90.000,E1 61.335} C_DIS
LIN {X 0.064,Y -289.629,Z 1616.330,A 0.000,B 0.000,C 90.000,E1 59.331} C_DIS
LIN {X -0.056,Y -281.248,Z 1616.318,A 0.000,B 0.000,C 90.000,E1 57.327} C_DIS
LIN {X -0.029,Y -272.483,Z 1616.307,A 0.000,B 0.000,C 90.000,E1 55.261} C_DIS
LIN {X -0.104,Y -260.655,Z 1616.291,A 0.000,B 0.000,C 90.000,E1 52.477} C_DIS
LIN {X 0.028,Y -247.855,Z 1616.273,A 0.000,B 0.000,C 90.000,E1 49.218} C_DIS
LIN {X -0.036,Y -237.581,Z 1616.257,A 0.000,B 0.000,C 90.000,E1 46.296} C_DIS
LIN {X -0.084,Y -227.044,Z 1616.238,A 0.000,B 0.000,C 90.000,E1 42.933} C_DIS
LIN {X 0.013,Y -218.544,Z 1616.221,A 0.000,B 0.000,C 90.000,E1 39.850} C_DIS
LIN {X -0.002,Y -210.817,Z 1616.204,A 0.000,B 0.000,C 90.000,E1 36.744} C_DIS
LIN {X 0.013,Y -203.912,Z 1616.187,A 0.000,B 0.000,C 90.000,E1 33.579} C_DIS
LIN {X -0.034,Y -197.699,Z 1616.169,A 0.000,B 0.000,C 90.000,E1 30.384} C_DIS
LIN {X -0.020,Y -192.209,Z 1616.151,A 0.000,B 0.000,C 90.000,E1 27.129} C_DIS
LIN {X 0.030,Y -187.482,Z 1616.132,A 0.000,B 0.000,C 90.000,E1 23.823} C_DIS
LIN {X -0.046,Y -182.498,Z 1616.109,A 0.000,B 0.000,C 90.000,E1 19.685} C_DIS
LIN {X -0.057,Y -178.401,Z 1616.086,A 0.000,B 0.000,C 90.000,E1 15.481} C_DIS
LIN {X -0.080,Y -174.963,Z 1616.062,A 0.000,B 0.000,C 90.000,E1 11.243} C_DIS
LIN {X -0.024,Y -172.074,Z 1616.034,A 0.000,B 0.000,C 90.000,E1 6.087} C_DIS
LIN {X -0.019,Y -170.257,Z 1616.005,A 0.000,B 0.000,C 90.000,E1 0.917} C_DIS
LIN {X 0.035,Y -171.223,Z 1615.930,A 0.000,B 0.000,C 90.000,E1 347.409} C_DIS
LIN {X 0.062,Y -174.246,Z 1615.901,A 0.000,B 0.000,C 90.000,E1 342.236} C_DIS
LIN {X -0.040,Y -177.228,Z 1615.882,A 0.000,B 0.000,C 90.000,E1 338.847} C_DIS
LIN {X 0.015,Y -181.103,Z 1615.864,A 0.000,B 0.000,C 90.000,E1 335.433} C_DIS
LIN {X -0.101,Y -185.814,Z 1615.845,A 0.000,B 0.000,C 90.000,E1 332.103} C_DIS
LIN {X 0.004,Y -191.405,Z 1615.826,A 0.000,B 0.000,C 90.000,E1 328.742} C_DIS
LIN {X -0.041,Y -197.731,Z 1615.808,A 0.000,B 0.000,C 90.000,E1 325.468} C_DIS
LIN {X 0.092,Y -204.842,Z 1615.790,A 0.000,B 0.000,C 90.000,E1 322.190} C_DIS
LIN {X 0.057,Y -212.846,Z 1615.772,A 0.000,B 0.000,C 90.000,E1 319.013} C_DIS
LIN {X 0.043,Y -221.891,Z 1615.755,A 0.000,B 0.000,C 90.000,E1 315.891} C_DIS
LIN {X -0.061,Y -231.948,Z 1615.738,A 0.000,B 0.000,C 90.000,E1 312.852} C_DIS
LIN {X 0.044,Y -238.859,Z 1615.728,A 0.000,B 0.000,C 90.000,E1 310.943} C_DIS
LIN {X -0.087,Y -248.155,Z 1615.715,A 0.000,B 0.000,C 90.000,E1 308.749} C_DIS
LIN {X -0.041,Y -256.804,Z 1615.705,A 0.000,B 0.000,C 90.000,E1 306.916} C_DIS
LIN {X 0.107,Y -268.423,Z 1615.693,A 0.000,B 0.000,C 90.000,E1 304.739} C_DIS
LIN {X 0.021,Y -279.015,Z 1615.683,A 0.000,B 0.000,C 90.000,E1 303.007} C_DIS
LIN {X 0.141,Y -297.786,Z 1615.668,A 0.000,B 0.000,C 90.000,E1 300.256} C_DIS
LIN {X -0.051,Y -312.615,Z 1615.657,A 0.000,B 0.000,C 90.000,E1 298.309} C_DIS
LIN {X 0.037,Y -327.522,Z 1615.646,A 0.000,B 0.000,C 90.000,E1 296.360} C_DIS
LIN {X 0.130,Y -339.680,Z 1615.638,A 0.000,B 0.000,C 90.000,E1 294.771} C_DIS
LIN {X -0.015,Y -353.979,Z 1615.627,A 0.000,B 0.000,C 90.000,E1 292.950} C_DIS
LIN {X 0.039,Y -370.927,Z 1615.616,A 0.000,B 0.000,C 90.000,E1 290.844} C_DIS
LIN {X -0.051,Y -380.176,Z 1615.609,A 0.000,B 0.000,C 90.000,E1 289.685} C_DIS
LIN {X 0.193,Y -386.553,Z 1615.604,A 0.000,B 0.000,C 90.000,E1 288.779} C_DIS
LIN {X 0.020,Y -392.502,Z 1615.600,A 0.000,B 0.000,C 90.000,E1 287.946} C_DIS
LIN {X 0.013,Y -397.815,Z 1615.595,A 0.000,B 0.000,C 90.000,E1 287.094} C_DIS
LIN {X -0.060,Y -402.418,Z 1615.590,A 0.000,B 0.000,C 90.000,E1 286.260} C_DIS
LIN {X -0.094,Y -406.138,Z 1615.586,A 0.000,B 0.000,C 90.000,E1 285.426} C_DIS
LIN {X 0.202,Y -408.147,Z 1615.583,A 0.000,B 0.000,C 90.000,E1 284.828} C_DIS
LIN {X 0.006,Y -409.801,Z 1615.579,A 0.000,B 0.000,C 90.000,E1 284.300} C_DIS
LIN {X -0.178,Y -411.089,Z 1615.576,A 0.000,B 0.000,C 90.000,E1 283.772} C_DIS
LIN {X 0.145,Y -411.815,Z 1615.573,A 0.000,B 0.000,C 90.000,E1 283.175} C_DIS
LIN {X -0.021,Y -412.148,Z 1615.570,A 0.000,B 0.000,C 90.000,E1 282.647} C_DIS
LIN {X -0.183,Y -411.978,Z 1615.567,A 0.000,B 0.000,C 90.000,E1 282.119} C_DIS
LIN {X 0.060,Y -411.294,Z 1615.564,A 0.000,B 0.000,C 90.000,E1 281.535} C_DIS
LIN {X -0.102,Y -410.064,Z 1615.561,A 0.000,B 0.000,C 90.000,E1 281.007} C_DIS
LIN {X 0.061,Y -408.266,Z 1615.558,A 0.000,B 0.000,C 90.000,E1 280.433} C_DIS
LIN {X -0.111,Y -405.787,Z 1615.555,A 0.000,B 0.000,C 90.000,E1 279.905} C_DIS
LIN {X -0.006,Y -404.329,Z 1615.553,A 0.000,B 0.000,C 90.000,E1 279.613} C_DIS
LIN {X 0.191,Y -400.790,Z 1615.550,A 0.000,B 0.000,C 90.000,E1 279.029} C_DIS
LIN {X -0.088,Y -396.690,Z 1615.547,A 0.000,B 0.000,C 90.000,E1 278.511} C_DIS
LIN {X 0.007,Y -392.014,Z 1615.544,A 0.000,B 0.000,C 90.000,E1 277.936} C_DIS
LIN {X 0.147,Y -386.743,Z 1615.541,A 0.000,B 0.000,C 90.000,E1 277.352} C_DIS
LIN {X -0.014,Y -381.063,Z 1615.538,A 0.000,B 0.000,C 90.000,E1 276.834} C_DIS
LIN {X 0.071,Y -375.232,Z 1615.535,A 0.000,B 0.000,C 90.000,E1 276.315} C_DIS
LIN {X 0.033,Y -366.001,Z 1615.531,A 0.000,B 0.000,C 90.000,E1 275.625} C_DIS
LIN {X -0.070,Y -359.596,Z 1615.529,A 0.000,B 0.000,C 90.000,E1 275.220} C_DIS
LIN {X 0.030,Y -353.143,Z 1615.527,A 0.000,B 0.000,C 90.000,E1 274.821} C_DIS
LIN {X 0.053,Y -343.453,Z 1615.524,A 0.000,B 0.000,C 90.000,E1 274.302} C_DIS
LIN {X 0.048,Y -333.715,Z 1615.521,A 0.000,B 0.000,C 90.000,E1 273.841} C_DIS
LIN {X 0.000,Y -324.114,Z 1615.519,A 0.000,B 0.000,C 90.000,E1 273.440} C_DIS
LIN {X -0.124,Y -314.177,Z 1615.517,A 0.000,B 0.000,C 90.000,E1 273.094} C_DIS
LIN {X -0.068,Y -303.780,Z 1615.515,A 0.000,B 0.000,C 90.000,E1 272.751} C_DIS
LIN {X 0.107,Y -296.469,Z 1615.514,A 0.000,B 0.000,C 90.000,E1 272.522} C_DIS
LIN {X 0.131,Y -288.782,Z 1615.513,A 0.000,B 0.000,C 90.000,E1 272.350} C_DIS
LIN {X 0.017,Y -280.612,Z 1615.512,A 0.000,B 0.000,C 90.000,E1 272.236} C_DIS
LIN {X 0.029,Y -265.844,Z 1615.511,A 0.000,B 0.000,C 90.000,E1 272.064} C_DIS
LIN {X -0.097,Y -249.891,Z 1615.511,A 0.000,B 0.000,C 90.000,E1 271.949} C_DIS
LIN {X 0.061,Y -229.883,Z 1615.510,A 0.000,B 0.000,C 90.000,E1 271.776} C_DIS
LIN {X -0.068,Y -221.786,Z 1615.510,A 0.000,B 0.000,C 90.000,E1 271.776} C_DIS
LIN {X 0.090,Y -181.305,Z 1615.510,A 0.000,B 0.000,C 90.000,E1 271.718} C_DIS
LIN {X 0.059,Y -181.563,Z 1615.500,A 0.000,B 0.000,C 90.000,E1 270.000} C_DIS
LIN {X 0.045,Y -180.854,Z 1615.472,A 0.000,B 0.000,C 90.000,E1 264.951} C_DIS
LIN {X -0.081,Y -178.964,Z 1615.444,A 0.000,B 0.000,C 90.000,E1 259.926} C_DIS
LIN {X -0.070,Y -177.914,Z 1615.434,A 0.000,B 0.000,C 90.000,E1 258.229} C_DIS
LIN {X -0.055,Y -175.551,Z 1615.411,A 0.000,B 0.000,C 90.000,E1 253.976} C_DIS
LIN {X -0.047,Y -172.282,Z 1615.387,A 0.000,B 0.000,C 90.000,E1 249.699} C_DIS
LIN {X -0.007,Y -171.761,Z 1615.382,A 0.000,B 0.000,C 90.000,E1 248.827} C_DIS
LIN {X 0.010,Y -167.361,Z 1615.354,A 0.000,B 0.000,C 90.000,E1 243.640} C_DIS
LIN {X -0.057,Y -166.750,Z 1615.349,A 0.000,B 0.000,C 90.000,E1 242.794} C_DIS
LIN {X 0.003,Y -162.730,Z 1615.324,A 0.000,B 0.000,C 90.000,E1 238.408} C_DIS
LIN {X 0.064,Y -161.421,Z 1615.315,A 0.000,B 0.000,C 90.000,E1 236.628} C_DIS
LIN {X 0.106,Y -157.413,Z 1615.290,A 0.000,B 0.000,C 90.000,E1 232.190} C_DIS
LIN {X 0.038,Y -155.415,Z 1615.275,A 0.000,B 0.000,C 90.000,E1 229.542} C_DIS
LIN {X -0.031,Y -151.742,Z 1615.250,A 0.000,B 0.000,C 90.000,E1 225.081} C_DIS
LIN {X -0.020,Y -149.940,Z 1615.235,A 0.000,B 0.000,C 90.000,E1 222.366} C_DIS
LIN {X 0.009,Y -146.787,Z 1615.210,A 0.000,B 0.000,C 90.000,E1 217.810} C_DIS
LIN {X -0.091,Y -145.360,Z 1615.195,A 0.000,B 0.000,C 90.000,E1 215.105} C_DIS
LIN {X 0.026,Y -142.429,Z 1615.164,A 0.000,B 0.000,C 90.000,E1 209.539} C_DIS
LIN {X 0.076,Y -141.417,Z 1615.149,A 0.000,B 0.000,C 90.000,E1 206.744} C_DIS
LIN {X 0.062,Y -139.361,Z 1615.113,A 0.000,B 0.000,C 90.000,E1 200.248} C_DIS
LIN {X 0.051,Y -138.804,Z 1615.097,A 0.000,B 0.000,C 90.000,E1 197.457} C_DIS
LIN {X -0.031,Y -138.350,Z 1615.056,A 0.000,B 0.000,C 90.000,E1 190.018} C_DIS
LIN {X -0.056,Y -139.545,Z 1615.004,A 0.000,B 0.000,C 90.000,E1 180.688} C_DIS
LIN {X 0.037,Y -141.248,Z 1614.973,A 0.000,B 0.000,C 90.000,E1 175.065} C_DIS
LIN {X -0.005,Y -142.618,Z 1614.957,A 0.000,B 0.000,C 90.000,E1 172.299} C_DIS
LIN {X -0.052,Y -144.935,Z 1614.932,A 0.000,B 0.000,C 90.000,E1 167.701} C_DIS
LIN {X 0.081,Y -147.564,Z 1614.911,A 0.000,B 0.000,C 90.000,E1 163.976} C_DIS
LIN {X -0.029,Y -150.171,Z 1614.891,A 0.000,B 0.000,C 90.000,E1 160.369} C_DIS
LIN {X -0.021,Y -153.546,Z 1614.871,A 0.000,B 0.000,C 90.000,E1 156.741} C_DIS
LIN {X 0.031,Y -156.964,Z 1614.851,A 0.000,B 0.000,C 90.000,E1 153.127} C_DIS
LIN {X -0.033,Y -161.072,Z 1614.831,A 0.000,B 0.000,C 90.000,E1 149.587} C_DIS
LIN {X 0.052,Y -163.179,Z 1614.821,A 0.000,B 0.000,C 90.000,E1 147.788} C_DIS
LIN {X 0.058,Y -167.600,Z 1614.802,A 0.000,B 0.000,C 90.000,E1 144.276} C_DIS
LIN {X -0.033,Y -171.428,Z 1614.787,A 0.000,B 0.000,C 90.000,E1 141.698} C_DIS
LIN {X 0.005,Y -176.347,Z 1614.768,A 0.000,B 0.000,C 90.000,E1 138.243} C_DIS
LIN {X 0.002,Y -180.638,Z 1614.754,A 0.000,B 0.000,C 90.000,E1 135.688} C_DIS
LIN {X -0.014,Y -186.040,Z 1614.735,A 0.000,B 0.000,C 90.000,E1 132.324} C_DIS
LIN {X 0.049,Y -190.676,Z 1614.721,A 0.000,B 0.000,C 90.000,E1 129.806} C_DIS
LIN {X 0.082,Y -196.428,Z 1614.703,A 0.000,B 0.000,C 90.000,E1 126.503} C_DIS
LIN {X 0.050,Y -201.212,Z 1614.689,A 0.000,B 0.000,C 90.000,E1 124.072} C_DIS
LIN {X 0.101,Y -205.531,Z 1614.676,A 0.000,B 0.000,C 90.000,E1 121.671} C_DIS
LIN {X 0.102,Y -324.793,Z 1614.676,A 0.000,B 0.000,C 90.000,E1 121.671} C_DIS
LIN {X 0.024,Y -329.203,Z 1614.675,A 0.000,B 0.000,C 90.000,E1 121.544} C_DIS
LIN {X -0.129,Y -332.561,Z 1614.674,A 0.000,B 0.000,C 90.000,E1 121.337} C_DIS
LIN {X -0.127,Y -336.233,Z 1614.672,A 0.000,B 0.000,C 90.000,E1 120.924} C_DIS
LIN {X 0.072,Y -338.109,Z 1614.670,A 0.000,B 0.000,C 90.000,E1 120.590} C_DIS
LIN {X -0.047,Y -340.840,Z 1614.667,A 0.000,B 0.000,C 90.000,E1 120.001} C_DIS
LIN {X -0.141,Y -352.880,Z 1614.651,A 0.000,B 0.000,C 90.000,E1 117.257} C_DIS
LIN {X 0.110,Y -366.372,Z 1614.636,A 0.000,B 0.000,C 90.000,E1 114.515} C_DIS
LIN {X -0.164,Y -379.685,Z 1614.623,A 0.000,B 0.000,C 90.000,E1 112.206} C_DIS
LIN {X -0.037,Y -394.331,Z 1614.610,A 0.000,B 0.000,C 90.000,E1 109.885} C_DIS
LIN {X -0.044,Y -410.413,Z 1614.598,A 0.000,B 0.000,C 90.000,E1 107.638} C_DIS
LIN {X 0.096,Y -428.041,Z 1614.586,A 0.000,B 0.000,C 90.000,E1 105.426} C_DIS
LIN {X 0.080,Y -447.277,Z 1614.574,A 0.000,B 0.000,C 90.000,E1 103.300} C_DIS
LIN {X 0.226,Y -467.383,Z 1614.563,A 0.000,B 0.000,C 90.000,E1 101.299} C_DIS
LIN {X 0.166,Y -490.648,Z 1614.552,A 0.000,B 0.000,C 90.000,E1 99.265} C_DIS
LIN {X -0.032,Y -495.897,Z 1614.549,A 0.000,B 0.000,C 90.000,E1 98.859} C_DIS
LIN {X 0.185,Y -498.137,Z 1614.548,A 0.000,B 0.000,C 90.000,E1 98.624} C_DIS
LIN {X -0.166,Y -499.838,Z 1614.547,A 0.000,B 0.000,C 90.000,E1 98.454} C_DIS
LIN {X 0.254,Y -501.341,Z 1614.546,A 0.000,B 0.000,C 90.000,E1 98.163} C_DIS
LIN {X 0.107,Y -502.457,Z 1614.544,A 0.000,B 0.000,C 90.000,E1 97.936} C_DIS
LIN {X -0.031,Y -503.764,Z 1614.542,A 0.000,B 0.000,C 90.000,E1 97.466} C_DIS
LIN {X 0.267,Y -504.021,Z 1614.539,A 0.000,B 0.000,C 90.000,E1 96.947} C_DIS
LIN {X 0.074,Y -503.271,Z 1614.536,A 0.000,B 0.000,C 90.000,E1 96.486} C_DIS
LIN {X -0.119,Y -501.387,Z 1614.533,A 0.000,B 0.000,C 90.000,E1 96.024} C_DIS
LIN {X 0.134,Y -498.186,Z 1614.531,A 0.000,B 0.000,C 90.000,E1 95.511} C_DIS
LIN {X 0.112,Y -484.852,Z 1614.520,A 0.000,B 0.000,C 90.000,E1 93.555} C_DIS
LIN {X 0.103,Y -474.788,Z 1614.511,A 0.000,B 0.000,C 90.000,E1 92.064} C_DIS
LIN {X 0.120,Y -466.058,Z 1614.505,A 0.000,B 0.000,C 90.000,E1 90.802} C_DIS
LIN {X -0.214,Y -455.200,Z 1614.496,A 0.000,B 0.000,C 90.000,E1 89.312} C_DIS
LIN {X -0.012,Y -445.810,Z 1614.489,A 0.000,B 0.000,C 90.000,E1 87.993} C_DIS
LIN {X 0.046,Y -435.954,Z 1614.482,A 0.000,B 0.000,C 90.000,E1 86.674} C_DIS
LIN {X -0.178,Y -421.913,Z 1614.471,A 0.000,B 0.000,C 90.000,E1 84.837} C_DIS
LIN {X 0.121,Y -400.662,Z 1614.454,A 0.000,B 0.000,C 90.000,E1 81.781} C_DIS
LIN {X -0.085,Y -381.073,Z 1614.437,A 0.000,B 0.000,C 90.000,E1 78.701} C_DIS
LIN {X 0.076,Y -365.995,Z 1614.423,A 0.000,B 0.000,C 90.000,E1 76.061} C_DIS
LIN {X 0.064,Y -353.027,Z 1614.409,A 0.000,B 0.000,C 90.000,E1 73.685} C_DIS
LIN {X -0.040,Y -339.030,Z 1614.394,A 0.000,B 0.000,C 90.000,E1 70.967} C_DIS
LIN {X 0.057,Y -326.994,Z 1614.380,A 0.000,B 0.000,C 90.000,E1 68.465} C_DIS
LIN {X 0.094,Y -315.728,Z 1614.366,A 0.000,B 0.000,C 90.000,E1 65.921} C_DIS
LIN {X 0.138,Y -304.032,Z 1614.350,A 0.000,B 0.000,C 90.000,E1 62.999} C_DIS
LIN {X -0.006,Y -296.314,Z 1614.339,A 0.000,B 0.000,C 90.000,E1 61.051} C_DIS
LIN {X -0.135,Y -289.632,Z 1614.330,A 0.000,B 0.000,C 90.000,E1 59.410} C_DIS
LIN {X -0.100,Y -281.245,Z 1614.319,A 0.000,B 0.000,C 90.000,E1 57.375} C_DIS
LIN {X -0.068,Y -272.435,Z 1614.307,A 0.000,B 0.000,C 90.000,E1 55.308} C_DIS
LIN {X 0.072,Y -260.574,Z 1614.292,A 0.000,B 0.000,C 90.000,E1 52.477} C_DIS
LIN {X 0.033,Y -247.793,Z 1614.274,A 0.000,B 0.000,C 90.000,E1 49.256} C_DIS
LIN {X 0.121,Y -237.548,Z 1614.257,A 0.000,B 0.000,C 90.000,E1 46.296} C_DIS
LIN {X 0.066,Y -227.039,Z 1614.239,A 0.000,B 0.000,C 90.000,E1 42.933} C_DIS
LIN {X 0.024,Y -218.561,Z 1614.222,A 0.000,B 0.000,C 90.000,E1 39.886} C_DIS
LIN {X -0.025,Y -210.852,Z 1614.204,A 0.000,B 0.000,C 90.000,E1 36.790} C_DIS
LIN {X -0.014,Y -203.965,Z 1614.187,A 0.000,B 0.000,C 90.000,E1 33.627} C_DIS
LIN {X 0.006,Y -197.769,Z 1614.169,A 0.000,B 0.000,C 90.000,E1 30.413} C_DIS
LIN {X -0.054,Y -192.310,Z 1614.151,A 0.000,B 0.000,C 90.000,E1 27.180} C_DIS
LIN {X -0.081,Y -187.586,Z 1614.133,A 0.000,B 0.000,C 90.000,E1 23.898} C_DIS
LIN {X 0.029,Y -182.625,Z 1614.109,A 0.000,B 0.000,C 90.000,E1 19.704} C_DIS
LIN {X 0.079,Y -178.527,Z 1614.086,A 0.000,B 0.000,C 90.000,E1 15.481} C_DIS
LIN {X 0.058,Y -175.101,Z 1614.063,A 0.000,B 0.000,C 90.000,E1 11.243} C_DIS
LIN {X -0.054,Y -172.236,Z 1614.034,A 0.000,B 0.000,C 90.000,E1 6.144} C_DIS
LIN {X -0.043,Y -170.432,Z 1614.005,A 0.000,B 0.000,C 90.000,E1 0.974} C_DIS
LIN {X 0.050,Y -171.423,Z 1613.930,A 0.000,B 0.000,C 90.000,E1 347.409} C_DIS
LIN {X 0.084,Y -174.444,Z 1613.901,A 0.000,B 0.000,C 90.000,E1 342.236} C_DIS
LIN {X -0.011,Y -177.448,Z 1613.882,A 0.000,B 0.000,C 90.000,E1 338.847} C_DIS
LIN {X 0.050,Y -181.312,Z 1613.864,A 0.000,B 0.000,C 90.000,E1 335.433} C_DIS
LIN {X -0.060,Y -186.011,Z 1613.845,A 0.000,B 0.000,C 90.000,E1 332.103} C_DIS
LIN {X 0.051,Y -191.564,Z 1613.826,A 0.000,B 0.000,C 90.000,E1 328.742} C_DIS
LIN {X 0.011,Y -197.884,Z 1613.808,A 0.000,B 0.000,C 90.000,E1 325.468} C_DIS
LIN {X -0.137,Y -204.970,Z 1613.790,A 0.000,B 0.000,C 90.000,E1 322.271} C_DIS
LIN {X -0.040,Y -212.956,Z 1613.772,A 0.000,B 0.000,C 90.000,E1 319.057} C_DIS
LIN {X 0.112,Y -221.955,Z 1613.755,A 0.000,B 0.000,C 90.000,E1 315.891} C_DIS
LIN {X 0.012,Y -231.945,Z 1613.738,A 0.000,B 0.000,C 90.000,E1 312.852} C_DIS
LIN {X -0.093,Y -240.299,Z 1613.726,A 0.000,B 0.000,C 90.000,E1 310.620} C_DIS
LIN {X -0.011,Y -249.731,Z 1613.713,A 0.000,B 0.000,C 90.000,E1 308.382} C_DIS
LIN {X -0.087,Y -258.525,Z 1613.703,A 0.000,B 0.000,C 90.000,E1 306.583} C_DIS
LIN {X 0.100,Y -270.328,Z 1613.691,A 0.000,B 0.000,C 90.000,E1 304.405} C_DIS
LIN {X 0.039,Y -281.116,Z 1613.682,A 0.000,B 0.000,C 90.000,E1 302.673} C_DIS
LIN {X 0.080,Y -302.547,Z 1613.665,A 0.000,B 0.000,C 90.000,E1 299.617} C_DIS
LIN {X 0.130,Y -317.444,Z 1613.654,A 0.000,B 0.000,C 90.000,E1 297.641} C_DIS
LIN {X 0.065,Y -329.836,Z 1613.645,A 0.000,B 0.000,C 90.000,E1 296.052} C_DIS
LIN {X -0.104,Y -341.927,Z 1613.636,A 0.000,B 0.000,C 90.000,E1 294.515} C_DIS
LIN {X 0.146,Y -358.665,Z 1613.624,A 0.000,B 0.000,C 90.000,E1 292.333} C_DIS
LIN {X -0.003,Y -370.805,Z 1613.616,A 0.000,B 0.000,C 90.000,E1 290.865} C_DIS
LIN {X 0.041,Y -380.111,Z 1613.609,A 0.000,B 0.000,C 90.000,E1 289.685} C_DIS
LIN {X -0.081,Y -386.527,Z 1613.605,A 0.000,B 0.000,C 90.000,E1 288.833} C_DIS
LIN {X 0.113,Y -392.472,Z 1613.600,A 0.000,B 0.000,C 90.000,E1 287.946} C_DIS
LIN {X 0.107,Y -397.849,Z 1613.595,A 0.000,B 0.000,C 90.000,E1 287.094} C_DIS
LIN {X 0.036,Y -402.506,Z 1613.590,A 0.000,B 0.000,C 90.000,E1 286.260} C_DIS
LIN {X 0.002,Y -406.299,Z 1613.586,A 0.000,B 0.000,C 90.000,E1 285.426} C_DIS
LIN {X -0.094,Y -408.333,Z 1613.583,A 0.000,B 0.000,C 90.000,E1 284.883} C_DIS
LIN {X 0.105,Y -410.010,Z 1613.579,A 0.000,B 0.000,C 90.000,E1 284.300} C_DIS
LIN {X -0.076,Y -411.238,Z 1613.576,A 0.000,B 0.000,C 90.000,E1 283.772} C_DIS
LIN {X -0.153,Y -412.087,Z 1613.573,A 0.000,B 0.000,C 90.000,E1 283.231} C_DIS
LIN {X 0.082,Y -412.411,Z 1613.570,A 0.000,B 0.000,C 90.000,E1 282.647} C_DIS
LIN {X -0.077,Y -412.286,Z 1613.567,A 0.000,B 0.000,C 90.000,E1 282.119} C_DIS
LIN {X 0.167,Y -411.592,Z 1613.564,A 0.000,B 0.000,C 90.000,E1 281.535} C_DIS
LIN {X 0.007,Y -410.466,Z 1613.561,A 0.000,B 0.000,C 90.000,E1 281.007} C_DIS
LIN {X 0.170,Y -408.689,Z 1613.558,A 0.000,B 0.000,C 90.000,E1 280.433} C_DIS
LIN {X 0.001,Y -406.253,Z 1613.555,A 0.000,B 0.000,C 90.000,E1 279.905} C_DIS
LIN {X 0.211,Y -403.157,Z 1613.552,A 0.000,B 0.000,C 90.000,E1 279.321} C_DIS
LIN {X -0.057,Y -399.363,Z 1613.549,A 0.000,B 0.000,C 90.000,E1 278.803} C_DIS
LIN {X 0.110,Y -395.031,Z 1613.546,A 0.000,B 0.000,C 90.000,E1 278.219} C_DIS
LIN {X -0.193,Y -390.070,Z 1613.543,A 0.000,B 0.000,C 90.000,E1 277.701} C_DIS
LIN {X -0.121,Y -384.441,Z 1613.539,A 0.000,B 0.000,C 90.000,E1 277.125} C_DIS
LIN {X -0.140,Y -378.698,Z 1613.537,A 0.000,B 0.000,C 90.000,E1 276.606} C_DIS
LIN {X 0.054,Y -372.694,Z 1613.534,A 0.000,B 0.000,C 90.000,E1 276.087} C_DIS
LIN {X 0.119,Y -366.511,Z 1613.531,A 0.000,B 0.000,C 90.000,E1 275.625} C_DIS
LIN {X -0.071,Y -357.029,Z 1613.528,A 0.000,B 0.000,C 90.000,E1 275.049} C_DIS
LIN {X 0.145,Y -347.296,Z 1613.525,A 0.000,B 0.000,C 90.000,E1 274.473} C_DIS
LIN {X 0.058,Y -337.657,Z 1613.522,A 0.000,B 0.000,C 90.000,E1 274.012} C_DIS
LIN {X 0.094,Y -324.623,Z 1613.519,A 0.000,B 0.000,C 90.000,E1 273.440} C_DIS
LIN {X -0.023,Y -314.667,Z 1613.517,A 0.000,B 0.000,C 90.000,E1 273.094} C_DIS
LIN {X 0.029,Y -304.222,Z 1613.515,A 0.000,B 0.000,C 90.000,E1 272.751} C_DIS
LIN {X -0.106,Y -296.940,Z 1613.514,A 0.000,B 0.000,C 90.000,E1 272.579} C_DIS
LIN {X -0.089,Y -289.169,Z 1613.513,A 0.000,B 0.000,C 90.000,E1 272.407} C_DIS
LIN {X 0.081,Y -281.046,Z 1613.512,A 0.000,B 0.000,C 90.000,E1 272.236} C_DIS
LIN {X 0.083,Y -266.558,Z 1613.512,A 0.000,B 0.000,C 90.000,E1 272.064} C_DIS
LIN {X -0.101,Y -257.266,Z 1613.511,A 0.000,B 0.000,C 90.000,E1 272.007} C_DIS
LIN {X -0.081,Y -233.147,Z 1613.510,A 0.000,B 0.000,C 90.000,E1 271.835} C_DIS
LIN {X -0.021,Y -222.056,Z 1613.510,A 0.000,B 0.000,C 90.000,E1 271.776} C_DIS
LIN {X -0.053,Y -181.302,Z 1613.510,A 0.000,B 0.000,C 90.000,E1 271.776} C_DIS
LIN {X 0.064,Y -181.564,Z 1613.500,A 0.000,B 0.000,C 90.000,E1 270.000} C_DIS
LIN {X 0.050,Y -180.854,Z 1613.472,A 0.000,B 0.000,C 90.000,E1 264.951} C_DIS
LIN {X -0.075,Y -178.966,Z 1613.444,A 0.000,B 0.000,C 90.000,E1 259.926} C_DIS
LIN {X -0.065,Y -177.915,Z 1613.434,A 0.000,B 0.000,C 90.000,E1 258.229} C_DIS
LIN {X -0.049,Y -175.552,Z 1613.411,A 0.000,B 0.000,C 90.000,E1 253.976} C_DIS
LIN {X -0.042,Y -172.284,Z 1613.387,A 0.000,B 0.000,C 90.000,E1 249.699} C_DIS
LIN {X -0.002,Y -171.762,Z 1613.382,A 0.000,B 0.000,C 90.000,E1 248.827} C_DIS
LIN {X 0.015,Y -167.362,Z 1613.354,A 0.000,B 0.000,C 90.000,E1 243.640} C_DIS
LIN {X -0.052,Y -166.751,Z 1613.349,A 0.000,B 0.000,C 90.000,E1 242.794} C_DIS
LIN {X 0.008,Y -162.731,Z 1613.324,A 0.000,B 0.000,C 90.000,E1 238.408} C_DIS
LIN {X 0.070,Y -161.422,Z 1613.315,A 0.000,B 0.000,C 90.000,E1 236.628} C_DIS
LIN {X -0.014,Y -157.414,Z 1613.290,A 0.000,B 0.000,C 90.000,E1 232.236} C_DIS
LIN {X 0.042,Y -155.416,Z 1613.275,A 0.000,B 0.000,C 90.000,E1 229.542} C_DIS
LIN {X -0.027,Y -151.744,Z 1613.250,A 0.000,B 0.000,C 90.000,E1 225.081} C_DIS
LIN {X -0.015,Y -149.942,Z 1613.235,A 0.000,B 0.000,C 90.000,E1 222.366} C_DIS
LIN {X 0.013,Y -146.788,Z 1613.210,A 0.000,B 0.000,C 90.000,E1 217.810} C_DIS
LIN {X -0.086,Y -145.361,Z 1613.195,A 0.000,B 0.000,C 90.000,E1 215.105} C_DIS
LIN {X 0.030,Y -142.430,Z 1613.164,A 0.000,B 0.000,C 90.000,E1 209.539} C_DIS
LIN {X -0.047,Y -141.418,Z 1613.149,A 0.000,B 0.000,C 90.000,E1 206.796} C_DIS
LIN {X -0.064,Y -139.361,Z 1613.113,A 0.000,B 0.000,C 90.000,E1 200.301} C_DIS
LIN {X 0.055,Y -138.804,Z 1613.097,A 0.000,B 0.000,C 90.000,E1 197.457} C_DIS
LIN {X -0.027,Y -138.350,Z 1613.056,A 0.000,B 0.000,C 90.000,E1 190.018} C_DIS
LIN {X -0.051,Y -139.545,Z 1613.004,A 0.000,B 0.000,C 90.000,E1 180.688} C_DIS
LIN {X 0.041,Y -141.248,Z 1612.973,A 0.000,B 0.000,C 90.000,E1 175.065} C_DIS
LIN {X 0.000,Y -142.617,Z 1612.957,A 0.000,B 0.000,C 90.000,E1 172.299} C_DIS
LIN {X -0.048,Y -144.933,Z 1612.932,A 0.000,B 0.000,C 90.000,E1 167.701} C_DIS
LIN {X -0.056,Y -147.563,Z 1612.911,A 0.000,B 0.000,C 90.000,E1 164.031} C_DIS
LIN {X -0.024,Y -150.169,Z 1612.891,A 0.000,B 0.000,C 90.000,E1 160.369} C_DIS
LIN {X -0.016,Y -153.545,Z 1612.871,A 0.000,B 0.000,C 90.000,E1 156.741} C_DIS
LIN {X 0.036,Y -156.961,Z 1612.851,A 0.000,B 0.000,C 90.000,E1 153.127} C_DIS
LIN {X -0.028,Y -161.069,Z 1612.831,A 0.000,B 0.000,C 90.000,E1 149.587} C_DIS
LIN {X 0.056,Y -163.177,Z 1612.821,A 0.000,B 0.000,C 90.000,E1 147.788} C_DIS
LIN {X 0.063,Y -167.598,Z 1612.802,A 0.000,B 0.000,C 90.000,E1 144.276} C_DIS
LIN {X -0.028,Y -171.426,Z 1612.787,A 0.000,B 0.000,C 90.000,E1 141.698} C_DIS
LIN {X 0.011,Y -176.345,Z 1612.768,A 0.000,B 0.000,C 90.000,E1 138.243} C_DIS
LIN {X 0.007,Y -180.636,Z 1612.754,A 0.000,B 0.000,C 90.000,E1 135.688} C_DIS
LIN {X -0.008,Y -186.037,Z 1612.735,A 0.000,B 0.000,C 90.000,E1 132.324} C_DIS
LIN {X 0.055,Y -190.673,Z 1612.721,A 0.000,B 0.000,C 90.000,E1 129.806} C_DIS
LIN {X 0.088,Y -196.424,Z 1612.703,A 0.000,B 0.000,C 90.000,E1 126.503} C_DIS
LIN {X 0.055,Y -201.210,Z 1612.689,A 0.000,B 0.000,C 90.000,E1 124.072} C_DIS
LIN {X -0.038,Y -205.453,Z 1612.676,A 0.000,B 0.000,C 90.000,E1 121.750} C_DIS
LIN {X 0.076,Y -324.064,Z 1612.676,A 0.000,B 0.000,C 90.000,E1 121.720} C_DIS
LIN {X -0.001,Y -327.063,Z 1612.676,A 0.000,B 0.000,C 90.000,E1 121.671} C_DIS
LIN {X 0.202,Y -330.481,Z 1612.675,A 0.000,B 0.000,C 90.000,E1 121.465} C_DIS
LIN {X -0.102,Y -334.034,Z 1612.673,A 0.000,B 0.000,C 90.000,E1 121.209} C_DIS
LIN {X 0.163,Y -337.621,Z 1612.671,A 0.000,B 0.000,C 90.000,E1 120.669} C_DIS
LIN {X 0.004,Y -339.204,Z 1612.669,A 0.000,B 0.000,C 90.000,E1 120.384} C_DIS
LIN {X 0.036,Y -352.486,Z 1612.652,A 0.000,B 0.000,C 90.000,E1 117.308} C_DIS
LIN {X 0.117,Y -365.939,Z 1612.637,A 0.000,B 0.000,C 90.000,E1 114.591} C_DIS
LIN {X -0.038,Y -380.957,Z 1612.622,A 0.000,B 0.000,C 90.000,E1 111.972} C_DIS
LIN {X -0.105,Y -395.732,Z 1612.609,A 0.000,B 0.000,C 90.000,E1 109.685} C_DIS
LIN {X 0.176,Y -411.951,Z 1612.597,A 0.000,B 0.000,C 90.000,E1 107.402} C_DIS
LIN {X -0.049,Y -429.728,Z 1612.585,A 0.000,B 0.000,C 90.000,E1 105.245} C_DIS
LIN {X 0.000,Y -449.085,Z 1612.573,A 0.000,B 0.000,C 90.000,E1 103.119} C_DIS
LIN {X 0.170,Y -469.244,Z 1612.562,A 0.000,B 0.000,C 90.000,E1 101.130} C_DIS
LIN {X -0.233,Y -492.559,Z 1612.551,A 0.000,B 0.000,C 90.000,E1 99.151} C_DIS
LIN {X 0.084,Y -497.568,Z 1612.548,A 0.000,B 0.000,C 90.000,E1 98.690} C_DIS
LIN {X 0.174,Y -499.472,Z 1612.547,A 0.000,B 0.000,C 90.000,E1 98.454} C_DIS
LIN {X 0.262,Y -500.924,Z 1612.546,A 0.000,B 0.000,C 90.000,E1 98.219} C_DIS
LIN {X 0.120,Y -502.108,Z 1612.544,A 0.000,B 0.000,C 90.000,E1 97.992} C_DIS
LIN {X 0.047,Y -502.962,Z 1612.543,A 0.000,B 0.000,C 90.000,E1 97.757} C_DIS
LIN {X -0.156,Y -503.831,Z 1612.540,A 0.000,B 0.000,C 90.000,E1 97.296} C_DIS
LIN {X 0.148,Y -503.689,Z 1612.538,A 0.000,B 0.000,C 90.000,E1 96.777} C_DIS
LIN {X -0.045,Y -502.511,Z 1612.535,A 0.000,B 0.000,C 90.000,E1 96.315} C_DIS
LIN {X -0.167,Y -501.479,Z 1612.534,A 0.000,B 0.000,C 90.000,E1 96.087} C_DIS
LIN {X -0.236,Y -500.079,Z 1612.532,A 0.000,B 0.000,C 90.000,E1 95.853} C_DIS
LIN {X 0.114,Y -485.042,Z 1612.520,A 0.000,B 0.000,C 90.000,E1 93.612} C_DIS
LIN {X 0.107,Y -475.015,Z 1612.512,A 0.000,B 0.000,C 90.000,E1 92.121} C_DIS
LIN {X 0.132,Y -466.304,Z 1612.505,A 0.000,B 0.000,C 90.000,E1 90.859} C_DIS
LIN {X -0.197,Y -455.448,Z 1612.496,A 0.000,B 0.000,C 90.000,E1 89.370} C_DIS
LIN {X 0.002,Y -446.073,Z 1612.489,A 0.000,B 0.000,C 90.000,E1 88.051} C_DIS
LIN {X 0.071,Y -436.248,Z 1612.482,A 0.000,B 0.000,C 90.000,E1 86.731} C_DIS
LIN {X -0.153,Y -422.171,Z 1612.472,A 0.000,B 0.000,C 90.000,E1 84.894} C_DIS
LIN {X 0.062,Y -402.759,Z 1612.456,A 0.000,B 0.000,C 90.000,E1 82.129} C_DIS
LIN {X -0.078,Y -383.021,Z 1612.439,A 0.000,B 0.000,C 90.000,E1 79.050} C_DIS
LIN {X 0.141,Y -367.856,Z 1612.425,A 0.000,B 0.000,C 90.000,E1 76.408} C_DIS
LIN {X 0.133,Y -356.441,Z 1612.413,A 0.000,B 0.000,C 90.000,E1 74.338} C_DIS
LIN {X 0.007,Y -342.291,Z 1612.398,A 0.000,B 0.000,C 90.000,E1 71.638} C_DIS
LIN {X 0.087,Y -331.656,Z 1612.386,A 0.000,B 0.000,C 90.000,E1 69.464} C_DIS
LIN {X -0.123,Y -318.557,Z 1612.370,A 0.000,B 0.000,C 90.000,E1 66.666} C_DIS
LIN {X -0.081,Y -305.415,Z 1612.352,A 0.000,B 0.000,C 90.000,E1 63.435} C_DIS
LIN {X 0.073,Y -297.743,Z 1612.341,A 0.000,B 0.000,C 90.000,E1 61.435} C_DIS
LIN {X -0.033,Y -291.095,Z 1612.332,A 0.000,B 0.000,C 90.000,E1 59.793} C_DIS
LIN {X -0.097,Y -284.192,Z 1612.323,A 0.000,B 0.000,C 90.000,E1 58.122} C_DIS
LIN {X -0.112,Y -276.985,Z 1612.313,A 0.000,B 0.000,C 90.000,E1 56.421} C_DIS
LIN {X -0.007,Y -268.017,Z 1612.302,A 0.000,B 0.000,C 90.000,E1 54.322} C_DIS
LIN {X 0.128,Y -257.688,Z 1612.288,A 0.000,B 0.000,C 90.000,E1 51.823} C_DIS
LIN {X -0.015,Y -245.180,Z 1612.270,A 0.000,B 0.000,C 90.000,E1 48.609} C_DIS
LIN {X -0.016,Y -234.035,Z 1612.252,A 0.000,B 0.000,C 90.000,E1 45.283} C_DIS
LIN {X -0.006,Y -223.874,Z 1612.233,A 0.000,B 0.000,C 90.000,E1 41.881} C_DIS
LIN {X -0.097,Y -215.730,Z 1612.216,A 0.000,B 0.000,C 90.000,E1 38.830} C_DIS
LIN {X -0.007,Y -208.271,Z 1612.198,A 0.000,B 0.000,C 90.000,E1 35.678} C_DIS
LIN {X 0.001,Y -201.709,Z 1612.181,A 0.000,B 0.000,C 90.000,E1 32.498} C_DIS
LIN {X -0.029,Y -195.747,Z 1612.163,A 0.000,B 0.000,C 90.000,E1 29.283} C_DIS
LIN {X -0.060,Y -190.595,Z 1612.145,A 0.000,B 0.000,C 90.000,E1 26.027} C_DIS
LIN {X -0.033,Y -186.153,Z 1612.126,A 0.000,B 0.000,C 90.000,E1 22.717} C_DIS
LIN {X -0.034,Y -181.478,Z 1612.103,A 0.000,B 0.000,C 90.000,E1 18.544} C_DIS
LIN {X 0.049,Y -177.600,Z 1612.080,A 0.000,B 0.000,C 90.000,E1 14.300} C_DIS
LIN {X -0.038,Y -174.463,Z 1612.056,A 0.000,B 0.000,C 90.000,E1 10.074} C_DIS
LIN {X -0.041,Y -171.564,Z 1612.023,A 0.000,B 0.000,C 90.000,E1 4.073} C_DIS
LIN {X -0.015,Y -170.971,Z 1611.940,A 0.000,B 0.000,C 90.000,E1 349.162} C_DIS
LIN {X 0.036,Y -173.464,Z 1611.911,A 0.000,B 0.000,C 90.000,E1 343.976} C_DIS
LIN {X 0.021,Y -176.828,Z 1611.887,A 0.000,B 0.000,C 90.000,E1 339.699} C_DIS
LIN {X 0.001,Y -180.497,Z 1611.868,A 0.000,B 0.000,C 90.000,E1 336.305} C_DIS
LIN {X 0.040,Y -184.942,Z 1611.850,A 0.000,B 0.000,C 90.000,E1 332.922} C_DIS
LIN {X -0.057,Y -190.257,Z 1611.831,A 0.000,B 0.000,C 90.000,E1 329.616} C_DIS
LIN {X 0.032,Y -196.397,Z 1611.813,A 0.000,B 0.000,C 90.000,E1 326.294} C_DIS
LIN {X 0.014,Y -203.241,Z 1611.795,A 0.000,B 0.000,C 90.000,E1 323.050} C_DIS
LIN {X 0.094,Y -210.972,Z 1611.777,A 0.000,B 0.000,C 90.000,E1 319.828} C_DIS
LIN {X 0.048,Y -219.683,Z 1611.760,A 0.000,B 0.000,C 90.000,E1 316.701} C_DIS
LIN {X 0.043,Y -229.360,Z 1611.742,A 0.000,B 0.000,C 90.000,E1 313.623} C_DIS
LIN {X 0.014,Y -238.804,Z 1611.728,A 0.000,B 0.000,C 90.000,E1 310.987} C_DIS
LIN {X 0.068,Y -247.989,Z 1611.715,A 0.000,B 0.000,C 90.000,E1 308.749} C_DIS
LIN {X -0.037,Y -256.572,Z 1611.705,A 0.000,B 0.000,C 90.000,E1 306.950} C_DIS
LIN {X -0.105,Y -268.133,Z 1611.693,A 0.000,B 0.000,C 90.000,E1 304.818} C_DIS
LIN {X 0.120,Y -280.984,Z 1611.682,A 0.000,B 0.000,C 90.000,E1 302.673} C_DIS
LIN {X -0.100,Y -302.397,Z 1611.665,A 0.000,B 0.000,C 90.000,E1 299.667} C_DIS
LIN {X -0.067,Y -317.303,Z 1611.654,A 0.000,B 0.000,C 90.000,E1 297.692} C_DIS
LIN {X -0.147,Y -329.679,Z 1611.645,A 0.000,B 0.000,C 90.000,E1 296.104} C_DIS
LIN {X -0.018,Y -341.782,Z 1611.636,A 0.000,B 0.000,C 90.000,E1 294.515} C_DIS
LIN {X -0.099,Y -358.565,Z 1611.624,A 0.000,B 0.000,C 90.000,E1 292.386} C_DIS
LIN {X 0.085,Y -370.697,Z 1611.616,A 0.000,B 0.000,C 90.000,E1 290.865} C_DIS
LIN {X 0.016,Y -377.821,Z 1611.611,A 0.000,B 0.000,C 90.000,E1 289.993} C_DIS
LIN {X -0.118,Y -384.388,Z 1611.606,A 0.000,B 0.000,C 90.000,E1 289.141} C_DIS
LIN {X 0.169,Y -390.547,Z 1611.601,A 0.000,B 0.000,C 90.000,E1 288.236} C_DIS
LIN {X 0.032,Y -396.137,Z 1611.597,A 0.000,B 0.000,C 90.000,E1 287.402} C_DIS
LIN {X 0.056,Y -401.110,Z 1611.592,A 0.000,B 0.000,C 90.000,E1 286.551} C_DIS
LIN {X 0.012,Y -405.240,Z 1611.587,A 0.000,B 0.000,C 90.000,E1 285.717} C_DIS
LIN {X -0.200,Y -407.498,Z 1611.584,A 0.000,B 0.000,C 90.000,E1 285.190} C_DIS
LIN {X -0.103,Y -408.491,Z 1611.583,A 0.000,B 0.000,C 90.000,E1 284.898} C_DIS
LIN {X 0.210,Y -410.159,Z 1611.580,A 0.000,B 0.000,C 90.000,E1 284.300} C_DIS
LIN {X 0.029,Y -411.478,Z 1611.577,A 0.000,B 0.000,C 90.000,E1 283.772} C_DIS
LIN {X -0.141,Y -412.306,Z 1611.573,A 0.000,B 0.000,C 90.000,E1 283.244} C_DIS
LIN {X 0.190,Y -412.691,Z 1611.570,A 0.000,B 0.000,C 90.000,E1 282.647} C_DIS
LIN {X 0.031,Y -412.603,Z 1611.567,A 0.000,B 0.000,C 90.000,E1 282.119} C_DIS
LIN {X -0.126,Y -411.985,Z 1611.564,A 0.000,B 0.000,C 90.000,E1 281.591} C_DIS
LIN {X 0.119,Y -410.840,Z 1611.561,A 0.000,B 0.000,C 90.000,E1 281.007} C_DIS
LIN {X -0.118,Y -409.101,Z 1611.558,A 0.000,B 0.000,C 90.000,E1 280.489} C_DIS
LIN {X 0.116,Y -406.753,Z 1611.555,A 0.000,B 0.000,C 90.000,E1 279.905} C_DIS
LIN {X -0.070,Y -403.724,Z 1611.552,A 0.000,B 0.000,C 90.000,E1 279.378} C_DIS
LIN {X 0.061,Y -399.965,Z 1611.549,A 0.000,B 0.000,C 90.000,E1 278.803} C_DIS
LIN {X -0.161,Y -395.603,Z 1611.546,A 0.000,B 0.000,C 90.000,E1 278.276} C_DIS
LIN {X -0.071,Y -390.684,Z 1611.543,A 0.000,B 0.000,C 90.000,E1 277.701} C_DIS
LIN {X -0.008,Y -385.045,Z 1611.540,A 0.000,B 0.000,C 90.000,E1 277.125} C_DIS
LIN {X -0.036,Y -379.280,Z 1611.537,A 0.000,B 0.000,C 90.000,E1 276.606} C_DIS
LIN {X 0.164,Y -373.295,Z 1611.534,A 0.000,B 0.000,C 90.000,E1 276.087} C_DIS
LIN {X -0.141,Y -367.081,Z 1611.531,A 0.000,B 0.000,C 90.000,E1 275.682} C_DIS
LIN {X 0.066,Y -357.642,Z 1611.528,A 0.000,B 0.000,C 90.000,E1 275.049} C_DIS
LIN {X -0.050,Y -348.004,Z 1611.525,A 0.000,B 0.000,C 90.000,E1 274.531} C_DIS
LIN {X -0.141,Y -338.266,Z 1611.522,A 0.000,B 0.000,C 90.000,E1 274.069} C_DIS
LIN {X -0.023,Y -328.329,Z 1611.520,A 0.000,B 0.000,C 90.000,E1 273.612} C_DIS
LIN {X 0.086,Y -318.516,Z 1611.518,A 0.000,B 0.000,C 90.000,E1 273.212} C_DIS
LIN {X -0.145,Y -305.123,Z 1611.516,A 0.000,B 0.000,C 90.000,E1 272.808} C_DIS
LIN {X -0.136,Y -294.101,Z 1611.514,A 0.000,B 0.000,C 90.000,E1 272.522} C_DIS
LIN {X -0.082,Y -282.326,Z 1611.513,A 0.000,B 0.000,C 90.000,E1 272.293} C_DIS
LIN {X -0.095,Y -267.973,Z 1611.512,A 0.000,B 0.000,C 90.000,E1 272.121} C_DIS
LIN {X 0.012,Y -252.579,Z 1611.511,A 0.000,B 0.000,C 90.000,E1 271.949} C_DIS
LIN {X -0.085,Y -231.189,Z 1611.510,A 0.000,B 0.000,C 90.000,E1 271.833} C_DIS
LIN {X 0.052,Y -225.647,Z 1611.510,A 0.000,B 0.000,C 90.000,E1 271.776} C_DIS
LIN {X 0.008,Y -218.330,Z 1611.510,A 0.000,B 0.000,C 90.000,E1 271.776} C_DIS
LIN {X -0.030,Y -181.301,Z 1611.510,A 0.000,B 0.000,C 90.000,E1 271.776} C_DIS
LIN {X -0.066,Y -181.566,Z 1611.500,A 0.000,B 0.000,C 90.000,E1 270.057} C_DIS
LIN {X -0.078,Y -180.858,Z 1611.472,A 0.000,B 0.000,C 90.000,E1 265.008} C_DIS
LIN {X -0.024,Y -178.970,Z 1611.444,A 0.000,B 0.000,C 90.000,E1 259.926} C_DIS
LIN {X -0.014,Y -177.927,Z 1611.435,A 0.000,B 0.000,C 90.000,E1 258.229} C_DIS
LIN {X 0.001,Y -175.564,Z 1611.411,A 0.000,B 0.000,C 90.000,E1 253.976} C_DIS
LIN {X 0.008,Y -172.294,Z 1611.387,A 0.000,B 0.000,C 90.000,E1 249.699} C_DIS
LIN {X -0.014,Y -171.773,Z 1611.382,A 0.000,B 0.000,C 90.000,E1 248.847} C_DIS
LIN {X -0.041,Y -168.700,Z 1611.363,A 0.000,B 0.000,C 90.000,E1 245.409} C_DIS
LIN {X -0.003,Y -166.765,Z 1611.349,A 0.000,B 0.000,C 90.000,E1 242.794} C_DIS
LIN {X 0.056,Y -162.745,Z 1611.325,A 0.000,B 0.000,C 90.000,E1 238.408} C_DIS
LIN {X -0.106,Y -161.434,Z 1611.315,A 0.000,B 0.000,C 90.000,E1 236.707} C_DIS
LIN {X -0.063,Y -157.428,Z 1611.290,A 0.000,B 0.000,C 90.000,E1 232.271} C_DIS
LIN {X -0.029,Y -155.433,Z 1611.275,A 0.000,B 0.000,C 90.000,E1 229.585} C_DIS
LIN {X 0.020,Y -151.755,Z 1611.250,A 0.000,B 0.000,C 90.000,E1 225.081} C_DIS
LIN {X 0.031,Y -149.955,Z 1611.235,A 0.000,B 0.000,C 90.000,E1 222.366} C_DIS
LIN {X 0.058,Y -146.798,Z 1611.210,A 0.000,B 0.000,C 90.000,E1 217.810} C_DIS
LIN {X -0.041,Y -145.374,Z 1611.195,A 0.000,B 0.000,C 90.000,E1 215.105} C_DIS
LIN {X 0.075,Y -142.436,Z 1611.164,A 0.000,B 0.000,C 90.000,E1 209.539} C_DIS
LIN {X -0.001,Y -141.427,Z 1611.149,A 0.000,B 0.000,C 90.000,E1 206.796} C_DIS
LIN {X -0.020,Y -139.364,Z 1611.113,A 0.000,B 0.000,C 90.000,E1 200.301} C_DIS
LIN {X -0.034,Y -138.808,Z 1611.097,A 0.000,B 0.000,C 90.000,E1 197.511} C_DIS
LIN {X 0.016,Y -138.350,Z 1611.056,A 0.000,B 0.000,C 90.000,E1 190.018} C_DIS
LIN {X -0.007,Y -139.542,Z 1611.004,A 0.000,B 0.000,C 90.000,E1 180.688} C_DIS
LIN {X -0.055,Y -141.240,Z 1610.973,A 0.000,B 0.000,C 90.000,E1 175.122} C_DIS
LIN {X 0.045,Y -142.610,Z 1610.957,A 0.000,B 0.000,C 90.000,E1 172.299} C_DIS
LIN {X -0.003,Y -144.923,Z 1610.932,A 0.000,B 0.000,C 90.000,E1 167.701} C_DIS
LIN {X -0.010,Y -147.552,Z 1610.911,A 0.000,B 0.000,C 90.000,E1 164.031} C_DIS
LIN {X 0.022,Y -150.155,Z 1610.891,A 0.000,B 0.000,C 90.000,E1 160.369} C_DIS
LIN {X 0.031,Y -153.526,Z 1610.871,A 0.000,B 0.000,C 90.000,E1 156.741} C_DIS
LIN {X 0.084,Y -156.944,Z 1610.851,A 0.000,B 0.000,C 90.000,E1 153.127} C_DIS
LIN {X 0.020,Y -161.047,Z 1610.831,A 0.000,B 0.000,C 90.000,E1 149.587} C_DIS
LIN {X 0.105,Y -163.157,Z 1610.821,A 0.000,B 0.000,C 90.000,E1 147.788} C_DIS
LIN {X -0.024,Y -167.574,Z 1610.802,A 0.000,B 0.000,C 90.000,E1 144.322} C_DIS
LIN {X 0.022,Y -171.404,Z 1610.787,A 0.000,B 0.000,C 90.000,E1 141.698} C_DIS
LIN {X 0.062,Y -176.319,Z 1610.768,A 0.000,B 0.000,C 90.000,E1 138.243} C_DIS
LIN {X -0.070,Y -180.607,Z 1610.754,A 0.000,B 0.000,C 90.000,E1 135.729} C_DIS
LIN {X 0.044,Y -186.009,Z 1610.735,A 0.000,B 0.000,C 90.000,E1 132.324} C_DIS
LIN {X -0.038,Y -190.643,Z 1610.721,A 0.000,B 0.000,C 90.000,E1 129.850} C_DIS
LIN {X 0.026,Y -196.394,Z 1610.703,A 0.000,B 0.000,C 90.000,E1 126.537} C_DIS
LIN {X -0.056,Y -201.183,Z 1610.689,A 0.000,B 0.000,C 90.000,E1 124.119} C_DIS
LIN {X -0.061,Y -205.373,Z 1610.677,A 0.000,B 0.000,C 90.000,E1 121.799} C_DIS
LIN {X -0.131,Y -323.511,Z 1610.677,A 0.000,B 0.000,C 90.000,E1 121.799} C_DIS
LIN {X 0.038,Y -325.124,Z 1610.676,A 0.000,B 0.000,C 90.000,E1 121.750} C_DIS
LIN {X 0.087,Y -327.526,Z 1610.676,A 0.000,B 0.000,C 90.000,E1 121.671} C_DIS
LIN {X -0.072,Y -330.840,Z 1610.675,A 0.000,B 0.000,C 90.000,E1 121.514} C_DIS
LIN {X 0.176,Y -334.474,Z 1610.673,A 0.000,B 0.000,C 90.000,E1 121.131} C_DIS
LIN {X -0.204,Y -337.999,Z 1610.670,A 0.000,B 0.000,C 90.000,E1 120.669} C_DIS
LIN {X 0.063,Y -340.721,Z 1610.667,A 0.000,B 0.000,C 90.000,E1 120.001} C_DIS
LIN {X -0.024,Y -352.746,Z 1610.651,A 0.000,B 0.000,C 90.000,E1 117.257} C_DIS
LIN {X 0.223,Y -366.231,Z 1610.636,A 0.000,B 0.000,C 90.000,E1 114.515} C_DIS
LIN {X -0.051,Y -379.535,Z 1610.623,A 0.000,B 0.000,C 90.000,E1 112.206} C_DIS
LIN {X 0.076,Y -394.170,Z 1610.610,A 0.000,B 0.000,C 90.000,E1 109.885} C_DIS
LIN {X 0.069,Y -410.241,Z 1610.598,A 0.000,B 0.000,C 90.000,E1 107.638} C_DIS
LIN {X 0.209,Y -427.857,Z 1610.586,A 0.000,B 0.000,C 90.000,E1 105.426} C_DIS
LIN {X 0.186,Y -447.092,Z 1610.574,A 0.000,B 0.000,C 90.000,E1 103.300} C_DIS
LIN {X -0.225,Y -467.194,Z 1610.563,A 0.000,B 0.000,C 90.000,E1 101.366} C_DIS
LIN {X -0.205,Y -490.427,Z 1610.552,A 0.000,B 0.000,C 90.000,E1 99.321} C_DIS
LIN {X 0.079,Y -495.675,Z 1610.549,A 0.000,B 0.000,C 90.000,E1 98.859} C_DIS
LIN {X -0.212,Y -497.910,Z 1610.548,A 0.000,B 0.000,C 90.000,E1 98.681} C_DIS
LIN {X 0.213,Y -499.758,Z 1610.547,A 0.000,B 0.000,C 90.000,E1 98.398} C_DIS
LIN {X 0.218,Y -501.156,Z 1610.546,A 0.000,B 0.000,C 90.000,E1 98.163} C_DIS
LIN {X 0.005,Y -503.004,Z 1610.543,A 0.000,B 0.000,C 90.000,E1 97.701} C_DIS
LIN {X -0.202,Y -503.719,Z 1610.540,A 0.000,B 0.000,C 90.000,E1 97.239} C_DIS
LIN {X 0.102,Y -503.429,Z 1610.537,A 0.000,B 0.000,C 90.000,E1 96.720} C_DIS
LIN {X -0.090,Y -502.087,Z 1610.535,A 0.000,B 0.000,C 90.000,E1 96.258} C_DIS
LIN {X -0.160,Y -500.953,Z 1610.533,A 0.000,B 0.000,C 90.000,E1 96.024} C_DIS
LIN {X 0.086,Y -497.712,Z 1610.531,A 0.000,B 0.000,C 90.000,E1 95.511} C_DIS
LIN {X 0.211,Y -486.091,Z 1610.521,A 0.000,B 0.000,C 90.000,E1 93.784} C_DIS
LIN {X 0.040,Y -474.398,Z 1610.511,A 0.000,B 0.000,C 90.000,E1 92.064} C_DIS
LIN {X 0.057,Y -465.673,Z 1610.505,A 0.000,B 0.000,C 90.000,E1 90.802} C_DIS
LIN {X 0.174,Y -454.804,Z 1610.496,A 0.000,B 0.000,C 90.000,E1 89.255} C_DIS
LIN {X -0.089,Y -445.401,Z 1610.489,A 0.000,B 0.000,C 90.000,E1 87.993} C_DIS
LIN {X -0.029,Y -435.545,Z 1610.481,A 0.000,B 0.000,C 90.000,E1 86.674} C_DIS
LIN {X 0.155,Y -421.453,Z 1610.471,A 0.000,B 0.000,C 90.000,E1 84.780} C_DIS
LIN {X -0.011,Y -402.088,Z 1610.456,A 0.000,B 0.000,C 90.000,E1 82.064} C_DIS
LIN {X 0.182,Y -384.141,Z 1610.440,A 0.000,B 0.000,C 90.000,E1 79.218} C_DIS
LIN {X -0.009,Y -368.939,Z 1610.426,A 0.000,B 0.000,C 90.000,E1 76.645} C_DIS
LIN {X 0.005,Y -357.476,Z 1610.414,A 0.000,B 0.000,C 90.000,E1 74.574} C_DIS
LIN {X -0.081,Y -343.291,Z 1610.399,A 0.000,B 0.000,C 90.000,E1 71.873} C_DIS
LIN {X 0.009,Y -331.084,Z 1610.385,A 0.000,B 0.000,C 90.000,E1 69.390} C_DIS
LIN {X 0.088,Y -318.015,Z 1610.370,A 0.000,B 0.000,C 90.000,E1 66.538} C_DIS
LIN {X -0.031,Y -304.897,Z 1610.352,A 0.000,B 0.000,C 90.000,E1 63.332} C_DIS
LIN {X -0.158,Y -297.214,Z 1610.341,A 0.000,B 0.000,C 90.000,E1 61.385} C_DIS
LIN {X 0.126,Y -290.546,Z 1610.332,A 0.000,B 0.000,C 90.000,E1 59.665} C_DIS
LIN {X 0.049,Y -283.602,Z 1610.322,A 0.000,B 0.000,C 90.000,E1 57.995} C_DIS
LIN {X 0.020,Y -276.359,Z 1610.313,A 0.000,B 0.000,C 90.000,E1 56.294} C_DIS
LIN {X 0.021,Y -265.852,Z 1610.299,A 0.000,B 0.000,C 90.000,E1 53.863} C_DIS
LIN {X 0.061,Y -255.583,Z 1610.286,A 0.000,B 0.000,C 90.000,E1 51.376} C_DIS
LIN {X -0.139,Y -243.311,Z 1610.267,A 0.000,B 0.000,C 90.000,E1 48.162} C_DIS
LIN {X -0.023,Y -232.381,Z 1610.249,A 0.000,B 0.000,C 90.000,E1 44.798} C_DIS
LIN {X 0.021,Y -223.480,Z 1610.232,A 0.000,B 0.000,C 90.000,E1 41.757} C_DIS
LIN {X 0.060,Y -215.380,Z 1610.215,A 0.000,B 0.000,C 90.000,E1 38.669} C_DIS
LIN {X 0.133,Y -207.965,Z 1610.198,A 0.000,B 0.000,C 90.000,E1 35.518} C_DIS
LIN {X 0.123,Y -201.448,Z 1610.180,A 0.000,B 0.000,C 90.000,E1 32.339} C_DIS
LIN {X -0.019,Y -195.557,Z 1610.162,A 0.000,B 0.000,C 90.000,E1 29.155} C_DIS
LIN {X -0.055,Y -190.452,Z 1610.144,A 0.000,B 0.000,C 90.000,E1 25.899} C_DIS
LIN {X -0.032,Y -186.063,Z 1610.125,A 0.000,B 0.000,C 90.000,E1 22.589} C_DIS
LIN {X -0.039,Y -181.451,Z 1610.102,A 0.000,B 0.000,C 90.000,E1 18.417} C_DIS
LIN {X 0.037,Y -177.597,Z 1610.079,A 0.000,B 0.000,C 90.000,E1 14.175} C_DIS
LIN {X -0.085,Y -174.525,Z 1610.055,A 0.000,B 0.000,C 90.000,E1 9.962} C_DIS
LIN {X -0.068,Y -171.675,Z 1610.022,A 0.000,B 0.000,C 90.000,E1 3.955} C_DIS
LIN {X -0.043,Y -172.222,Z 1609.925,A 0.000,B 0.000,C 90.000,E1 346.589} C_DIS
LIN {X -0.087,Y -174.844,Z 1609.901,A 0.000,B 0.000,C 90.000,E1 342.308} C_DIS
LIN {X 0.047,Y -177.893,Z 1609.883,A 0.000,B 0.000,C 90.000,E1 338.847} C_DIS
LIN {X -0.045,Y -181.743,Z 1609.864,A 0.000,B 0.000,C 90.000,E1 335.485} C_DIS
LIN {X 0.023,Y -186.408,Z 1609.845,A 0.000,B 0.000,C 90.000,E1 332.103} C_DIS
LIN {X -0.018,Y -191.877,Z 1609.827,A 0.000,B 0.000,C 90.000,E1 328.791} C_DIS
LIN {X -0.045,Y -198.194,Z 1609.808,A 0.000,B 0.000,C 90.000,E1 325.515} C_DIS
LIN {X -0.020,Y -205.217,Z 1609.790,A 0.000,B 0.000,C 90.000,E1 322.271} C_DIS
LIN {X -0.052,Y -213.143,Z 1609.773,A 0.000,B 0.000,C 90.000,E1 319.094} C_DIS
LIN {X -0.064,Y -222.079,Z 1609.755,A 0.000,B 0.000,C 90.000,E1 315.972} C_DIS
LIN {X -0.011,Y -231.945,Z 1609.738,A 0.000,B 0.000,C 90.000,E1 312.894} C_DIS
LIN {X 0.060,Y -240.208,Z 1609.726,A 0.000,B 0.000,C 90.000,E1 310.620} C_DIS
LIN {X 0.146,Y -247.873,Z 1609.715,A 0.000,B 0.000,C 90.000,E1 308.749} C_DIS
LIN {X 0.041,Y -256.452,Z 1609.705,A 0.000,B 0.000,C 90.000,E1 306.950} C_DIS
LIN {X -0.026,Y -267.977,Z 1609.693,A 0.000,B 0.000,C 90.000,E1 304.818} C_DIS
LIN {X 0.048,Y -280.842,Z 1609.682,A 0.000,B 0.000,C 90.000,E1 302.704} C_DIS
LIN {X -0.027,Y -299.774,Z 1609.667,A 0.000,B 0.000,C 90.000,E1 300.001} C_DIS
LIN {X -0.038,Y -314.672,Z 1609.656,A 0.000,B 0.000,C 90.000,E1 298.025} C_DIS
LIN {X -0.002,Y -327.081,Z 1609.647,A 0.000,B 0.000,C 90.000,E1 296.411} C_DIS
LIN {X 0.078,Y -339.261,Z 1609.638,A 0.000,B 0.000,C 90.000,E1 294.823} C_DIS
LIN {X -0.049,Y -356.025,Z 1609.626,A 0.000,B 0.000,C 90.000,E1 292.695} C_DIS
LIN {X 0.087,Y -368.202,Z 1609.618,A 0.000,B 0.000,C 90.000,E1 291.173} C_DIS
LIN {X 0.103,Y -377.728,Z 1609.611,A 0.000,B 0.000,C 90.000,E1 289.993} C_DIS
LIN {X -0.030,Y -384.369,Z 1609.606,A 0.000,B 0.000,C 90.000,E1 289.141} C_DIS
LIN {X -0.113,Y -390.540,Z 1609.602,A 0.000,B 0.000,C 90.000,E1 288.290} C_DIS
LIN {X 0.121,Y -396.154,Z 1609.597,A 0.000,B 0.000,C 90.000,E1 287.402} C_DIS
LIN {X 0.032,Y -401.180,Z 1609.592,A 0.000,B 0.000,C 90.000,E1 286.567} C_DIS
LIN {X 0.104,Y -405.373,Z 1609.587,A 0.000,B 0.000,C 90.000,E1 285.717} C_DIS
LIN {X -0.105,Y -407.690,Z 1609.584,A 0.000,B 0.000,C 90.000,E1 285.190} C_DIS
LIN {X -0.092,Y -410.391,Z 1609.580,A 0.000,B 0.000,C 90.000,E1 284.356} C_DIS
LIN {X 0.125,Y -411.685,Z 1609.577,A 0.000,B 0.000,C 90.000,E1 283.772} C_DIS
LIN {X -0.042,Y -412.546,Z 1609.573,A 0.000,B 0.000,C 90.000,E1 283.244} C_DIS
LIN {X -0.112,Y -412.995,Z 1609.570,A 0.000,B 0.000,C 90.000,E1 282.703} C_DIS
LIN {X 0.133,Y -412.881,Z 1609.567,A 0.000,B 0.000,C 90.000,E1 282.119} C_DIS
LIN {X -0.023,Y -412.328,Z 1609.564,A 0.000,B 0.000,C 90.000,E1 281.591} C_DIS
LIN {X 0.224,Y -411.214,Z 1609.561,A 0.000,B 0.000,C 90.000,E1 281.007} C_DIS
LIN {X -0.013,Y -409.513,Z 1609.558,A 0.000,B 0.000,C 90.000,E1 280.489} C_DIS
LIN {X -0.178,Y -407.194,Z 1609.555,A 0.000,B 0.000,C 90.000,E1 279.962} C_DIS
LIN {X 0.040,Y -404.220,Z 1609.552,A 0.000,B 0.000,C 90.000,E1 279.378} C_DIS
LIN {X 0.173,Y -400.491,Z 1609.549,A 0.000,B 0.000,C 90.000,E1 278.803} C_DIS
LIN {X -0.047,Y -396.173,Z 1609.546,A 0.000,B 0.000,C 90.000,E1 278.276} C_DIS
LIN {X 0.045,Y -391.272,Z 1609.543,A 0.000,B 0.000,C 90.000,E1 277.701} C_DIS
LIN {X 0.110,Y -385.677,Z 1609.540,A 0.000,B 0.000,C 90.000,E1 277.125} C_DIS
LIN {X 0.064,Y -379.850,Z 1609.537,A 0.000,B 0.000,C 90.000,E1 276.606} C_DIS
LIN {X -0.100,Y -373.866,Z 1609.534,A 0.000,B 0.000,C 90.000,E1 276.144} C_DIS
LIN {X -0.001,Y -367.761,Z 1609.532,A 0.000,B 0.000,C 90.000,E1 275.682} C_DIS
LIN {X -0.052,Y -361.430,Z 1609.529,A 0.000,B 0.000,C 90.000,E1 275.277} C_DIS
LIN {X 0.070,Y -351.826,Z 1609.526,A 0.000,B 0.000,C 90.000,E1 274.702} C_DIS
LIN {X -0.147,Y -342.143,Z 1609.523,A 0.000,B 0.000,C 90.000,E1 274.245} C_DIS
LIN {X -0.061,Y -332.354,Z 1609.521,A 0.000,B 0.000,C 90.000,E1 273.784} C_DIS
LIN {X -0.089,Y -322.359,Z 1609.519,A 0.000,B 0.000,C 90.000,E1 273.383} C_DIS
LIN {X -0.118,Y -312.507,Z 1609.517,A 0.000,B 0.000,C 90.000,E1 273.037} C_DIS
LIN {X 0.086,Y -302.617,Z 1609.515,A 0.000,B 0.000,C 90.000,E1 272.694} C_DIS
LIN {X -0.017,Y -295.048,Z 1609.514,A 0.000,B 0.000,C 90.000,E1 272.522} C_DIS
LIN {X 0.010,Y -283.270,Z 1609.513,A 0.000,B 0.000,C 90.000,E1 272.293} C_DIS
LIN {X -0.025,Y -269.038,Z 1609.512,A 0.000,B 0.000,C 90.000,E1 272.121} C_DIS
LIN {X 0.080,Y -253.794,Z 1609.511,A 0.000,B 0.000,C 90.000,E1 271.949} C_DIS
LIN {X -0.105,Y -229.103,Z 1609.510,A 0.000,B 0.000,C 90.000,E1 271.833} C_DIS
LIN {X 0.077,Y -224.994,Z 1609.510,A 0.000,B 0.000,C 90.000,E1 271.776} C_DIS
LIN {X 0.025,Y -181.299,Z 1609.510,A 0.000,B 0.000,C 90.000,E1 271.776} C_DIS
LIN {X -0.012,Y -181.568,Z 1609.500,A 0.000,B 0.000,C 90.000,E1 270.057} C_DIS
LIN {X -0.025,Y -180.862,Z 1609.472,A 0.000,B 0.000,C 90.000,E1 265.008} C_DIS
LIN {X 0.029,Y -178.975,Z 1609.444,A 0.000,B 0.000,C 90.000,E1 259.926} C_DIS
LIN {X 0.039,Y -177.939,Z 1609.435,A 0.000,B 0.000,C 90.000,E1 258.229} C_DIS
LIN {X 0.054,Y -175.578,Z 1609.411,A 0.000,B 0.000,C 90.000,E1 253.976} C_DIS
LIN {X 0.060,Y -172.305,Z 1609.387,A 0.000,B 0.000,C 90.000,E1 249.699} C_DIS
LIN {X 0.038,Y -171.783,Z 1609.383,A 0.000,B 0.000,C 90.000,E1 248.847} C_DIS
LIN {X -0.016,Y -169.449,Z 1609.368,A 0.000,B 0.000,C 90.000,E1 246.282} C_DIS
LIN {X -0.028,Y -166.779,Z 1609.349,A 0.000,B 0.000,C 90.000,E1 242.820} C_DIS
LIN {X -0.032,Y -162.759,Z 1609.325,A 0.000,B 0.000,C 90.000,E1 238.456} C_DIS
LIN {X -0.056,Y -161.448,Z 1609.315,A 0.000,B 0.000,C 90.000,E1 236.707} C_DIS
LIN {X -0.014,Y -157.442,Z 1609.290,A 0.000,B 0.000,C 90.000,E1 232.271} C_DIS
LIN {X 0.020,Y -155.450,Z 1609.276,A 0.000,B 0.000,C 90.000,E1 229.585} C_DIS
LIN {X 0.068,Y -151.768,Z 1609.251,A 0.000,B 0.000,C 90.000,E1 225.081} C_DIS
LIN {X -0.022,Y -149.971,Z 1609.236,A 0.000,B 0.000,C 90.000,E1 222.405} C_DIS
LIN {X -0.010,Y -146.808,Z 1609.210,A 0.000,B 0.000,C 90.000,E1 217.855} C_DIS
LIN {X 0.006,Y -145.386,Z 1609.195,A 0.000,B 0.000,C 90.000,E1 215.105} C_DIS
LIN {X -0.002,Y -142.443,Z 1609.164,A 0.000,B 0.000,C 90.000,E1 209.589} C_DIS
LIN {X -0.020,Y -141.436,Z 1609.149,A 0.000,B 0.000,C 90.000,E1 206.821} C_DIS
LIN {X 0.025,Y -139.367,Z 1609.113,A 0.000,B 0.000,C 90.000,E1 200.301} C_DIS
LIN {X 0.012,Y -138.813,Z 1609.097,A 0.000,B 0.000,C 90.000,E1 197.511} C_DIS
LIN {X 0.062,Y -138.351,Z 1609.056,A 0.000,B 0.000,C 90.000,E1 190.018} C_DIS
LIN {X 0.039,Y -139.539,Z 1609.004,A 0.000,B 0.000,C 90.000,E1 180.688} C_DIS
LIN {X -0.009,Y -141.231,Z 1608.973,A 0.000,B 0.000,C 90.000,E1 175.122} C_DIS
LIN {X -0.050,Y -142.603,Z 1608.957,A 0.000,B 0.000,C 90.000,E1 172.356} C_DIS
LIN {X 0.045,Y -144.911,Z 1608.932,A 0.000,B 0.000,C 90.000,E1 167.701} C_DIS
LIN {X 0.037,Y -147.540,Z 1608.911,A 0.000,B 0.000,C 90.000,E1 164.031} C_DIS
LIN {X 0.070,Y -150.140,Z 1608.891,A 0.000,B 0.000,C 90.000,E1 160.369} C_DIS
LIN {X -0.061,Y -153.507,Z 1608.871,A 0.000,B 0.000,C 90.000,E1 156.794} C_DIS
LIN {X 0.002,Y -157.872,Z 1608.846,A 0.000,B 0.000,C 90.000,E1 152.281} C_DIS
LIN {X -0.043,Y -162.158,Z 1608.826,A 0.000,B 0.000,C 90.000,E1 148.742} C_DIS
LIN {X 0.071,Y -166.365,Z 1608.807,A 0.000,B 0.000,C 90.000,E1 145.182} C_DIS
LIN {X -0.060,Y -171.382,Z 1608.787,A 0.000,B 0.000,C 90.000,E1 141.743} C_DIS
LIN {X -0.017,Y -176.291,Z 1608.768,A 0.000,B 0.000,C 90.000,E1 138.286} C_DIS
LIN {X -0.017,Y -180.578,Z 1608.754,A 0.000,B 0.000,C 90.000,E1 135.729} C_DIS
LIN {X -0.038,Y -185.979,Z 1608.735,A 0.000,B 0.000,C 90.000,E1 132.366} C_DIS
LIN {X 0.018,Y -190.612,Z 1608.721,A 0.000,B 0.000,C 90.000,E1 129.850} C_DIS
LIN {X -0.075,Y -196.362,Z 1608.703,A 0.000,B 0.000,C 90.000,E1 126.583} C_DIS
LIN {X 0.001,Y -201.156,Z 1608.690,A 0.000,B 0.000,C 90.000,E1 124.119} C_DIS
LIN {X 0.068,Y -205.302,Z 1608.677,A 0.000,B 0.000,C 90.000,E1 121.799} C_DIS
LIN {X 0.073,Y -323.931,Z 1608.677,A 0.000,B 0.000,C 90.000,E1 121.799} C_DIS
LIN {X -0.099,Y -327.922,Z 1608.676,A 0.000,B 0.000,C 90.000,E1 121.720} C_DIS
LIN {X -0.049,Y -331.154,Z 1608.675,A 0.000,B 0.000,C 90.000,E1 121.514} C_DIS
LIN {X 0.031,Y -334.827,Z 1608.673,A 0.000,B 0.000,C 90.000,E1 121.131} C_DIS
LIN {X -0.054,Y -338.293,Z 1608.670,A 0.000,B 0.000,C 90.000,E1 120.590} C_DIS
LIN {X -0.030,Y -352.966,Z 1608.651,A 0.000,B 0.000,C 90.000,E1 117.206} C_DIS
LIN {X -0.103,Y -366.481,Z 1608.636,A 0.000,B 0.000,C 90.000,E1 114.515} C_DIS
LIN {X -0.031,Y -379.810,Z 1608.623,A 0.000,B 0.000,C 90.000,E1 112.153} C_DIS
LIN {X -0.127,Y -394.475,Z 1608.610,A 0.000,B 0.000,C 90.000,E1 109.866} C_DIS
LIN {X 0.119,Y -410.577,Z 1608.598,A 0.000,B 0.000,C 90.000,E1 107.583} C_DIS
LIN {X -0.140,Y -428.229,Z 1608.586,A 0.000,B 0.000,C 90.000,E1 105.426} C_DIS
LIN {X -0.164,Y -447.494,Z 1608.574,A 0.000,B 0.000,C 90.000,E1 103.300} C_DIS
LIN {X -0.013,Y -467.608,Z 1608.563,A 0.000,B 0.000,C 90.000,E1 101.299} C_DIS
LIN {X -0.044,Y -490.854,Z 1608.551,A 0.000,B 0.000,C 90.000,E1 99.265} C_DIS
LIN {X -0.242,Y -496.077,Z 1608.549,A 0.000,B 0.000,C 90.000,E1 98.859} C_DIS
LIN {X -0.039,Y -498.171,Z 1608.548,A 0.000,B 0.000,C 90.000,E1 98.624} C_DIS
LIN {X -0.184,Y -499.976,Z 1608.547,A 0.000,B 0.000,C 90.000,E1 98.398} C_DIS
LIN {X 0.241,Y -501.326,Z 1608.545,A 0.000,B 0.000,C 90.000,E1 98.106} C_DIS
LIN {X 0.028,Y -503.011,Z 1608.542,A 0.000,B 0.000,C 90.000,E1 97.644} C_DIS
LIN {X -0.177,Y -503.593,Z 1608.540,A 0.000,B 0.000,C 90.000,E1 97.182} C_DIS
LIN {X 0.127,Y -503.171,Z 1608.537,A 0.000,B 0.000,C 90.000,E1 96.663} C_DIS
LIN {X -0.065,Y -501.680,Z 1608.534,A 0.000,B 0.000,C 90.000,E1 96.201} C_DIS
LIN {X -0.136,Y -500.454,Z 1608.533,A 0.000,B 0.000,C 90.000,E1 95.967} C_DIS
LIN {X -0.112,Y -487.204,Z 1608.522,A 0.000,B 0.000,C 90.000,E1 94.012} C_DIS
LIN {X 0.221,Y -475.535,Z 1608.513,A 0.000,B 0.000,C 90.000,E1 92.236} C_DIS
LIN {X -0.221,Y -466.882,Z 1608.506,A 0.000,B 0.000,C 90.000,E1 91.031} C_DIS
LIN {X -0.077,Y -456.061,Z 1608.497,A 0.000,B 0.000,C 90.000,E1 89.484} C_DIS
LIN {X -0.112,Y -444.789,Z 1608.488,A 0.000,B 0.000,C 90.000,E1 87.936} C_DIS
LIN {X -0.061,Y -434.918,Z 1608.481,A 0.000,B 0.000,C 90.000,E1 86.617} C_DIS
LIN {X 0.109,Y -420.808,Z 1608.471,A 0.000,B 0.000,C 90.000,E1 84.723} C_DIS
LIN {X -0.074,Y -401.493,Z 1608.456,A 0.000,B 0.000,C 90.000,E1 82.008} C_DIS
LIN {X 0.102,Y -383.595,Z 1608.440,A 0.000,B 0.000,C 90.000,E1 79.162} C_DIS
LIN {X -0.104,Y -368.407,Z 1608.425,A 0.000,B 0.000,C 90.000,E1 76.589} C_DIS
LIN {X -0.101,Y -356.968,Z 1608.414,A 0.000,B 0.000,C 90.000,E1 74.519} C_DIS
LIN {X 0.125,Y -342.786,Z 1608.399,A 0.000,B 0.000,C 90.000,E1 71.764} C_DIS
LIN {X -0.124,Y -330.567,Z 1608.385,A 0.000,B 0.000,C 90.000,E1 69.337} C_DIS
LIN {X -0.119,Y -316.165,Z 1608.368,A 0.000,B 0.000,C 90.000,E1 66.177} C_DIS
LIN {X -0.056,Y -304.425,Z 1608.351,A 0.000,B 0.000,C 90.000,E1 63.256} C_DIS
LIN {X 0.085,Y -295.411,Z 1608.339,A 0.000,B 0.000,C 90.000,E1 60.923} C_DIS
LIN {X -0.074,Y -287.279,Z 1608.327,A 0.000,B 0.000,C 90.000,E1 58.948} C_DIS
LIN {X -0.087,Y -278.723,Z 1608.316,A 0.000,B 0.000,C 90.000,E1 56.914} C_DIS
LIN {X 0.047,Y -269.719,Z 1608.305,A 0.000,B 0.000,C 90.000,E1 54.815} C_DIS
LIN {X 0.112,Y -257.875,Z 1608.289,A 0.000,B 0.000,C 90.000,E1 51.984} C_DIS
LIN {X -0.032,Y -245.429,Z 1608.271,A 0.000,B 0.000,C 90.000,E1 48.771} C_DIS
LIN {X -0.024,Y -234.290,Z 1608.252,A 0.000,B 0.000,C 90.000,E1 45.445} C_DIS
LIN {X -0.098,Y -225.270,Z 1608.236,A 0.000,B 0.000,C 90.000,E1 42.447} C_DIS
LIN {X -0.008,Y -217.012,Z 1608.219,A 0.000,B 0.000,C 90.000,E1 39.358} C_DIS
LIN {X 0.069,Y -209.477,Z 1608.201,A 0.000,B 0.000,C 90.000,E1 36.217} C_DIS
LIN {X -0.072,Y -202.773,Z 1608.184,A 0.000,B 0.000,C 90.000,E1 33.086} C_DIS
LIN {X -0.077,Y -196.783,Z 1608.166,A 0.000,B 0.000,C 90.000,E1 29.873} C_DIS
LIN {X -0.080,Y -191.540,Z 1608.148,A 0.000,B 0.000,C 90.000,E1 26.616} C_DIS
LIN {X 0.050,Y -187.020,Z 1608.129,A 0.000,B 0.000,C 90.000,E1 23.281} C_DIS
LIN {X -0.032,Y -182.294,Z 1608.106,A 0.000,B 0.000,C 90.000,E1 19.141} C_DIS
LIN {X -0.098,Y -178.320,Z 1608.083,A 0.000,B 0.000,C 90.000,E1 14.954} C_DIS
LIN {X 0.051,Y -175.120,Z 1608.059,A 0.000,B 0.000,C 90.000,E1 10.658} C_DIS
LIN {X -0.061,Y -172.106,Z 1608.026,A 0.000,B 0.000,C 90.000,E1 4.702} C_DIS
LIN {X -0.043,Y -170.411,Z 1607.993,A 0.000,B 0.000,C 90.000,E1 358.682} C_DIS
LIN {X 0.055,Y -171.722,Z 1607.935,A 0.000,B 0.000,C 90.000,E1 348.285} C_DIS
LIN {X 0.007,Y -174.429,Z 1607.906,A 0.000,B 0.000,C 90.000,E1 343.142} C_DIS
LIN {X -0.089,Y -178.110,Z 1607.883,A 0.000,B 0.000,C 90.000,E1 338.901} C_DIS
LIN {X -0.009,Y -181.960,Z 1607.864,A 0.000,B 0.000,C 90.000,E1 335.485} C_DIS
LIN {X 0.066,Y -186.598,Z 1607.845,A 0.000,B 0.000,C 90.000,E1 332.103} C_DIS
LIN {X 0.030,Y -192.036,Z 1607.827,A 0.000,B 0.000,C 90.000,E1 328.791} C_DIS
LIN {X 0.010,Y -198.340,Z 1607.808,A 0.000,B 0.000,C 90.000,E1 325.515} C_DIS
LIN {X 0.039,Y -205.323,Z 1607.790,A 0.000,B 0.000,C 90.000,E1 322.271} C_DIS
LIN {X 0.014,Y -213.237,Z 1607.773,A 0.000,B 0.000,C 90.000,E1 319.094} C_DIS
LIN {X 0.005,Y -222.119,Z 1607.755,A 0.000,B 0.000,C 90.000,E1 315.972} C_DIS
LIN {X -0.096,Y -231.938,Z 1607.738,A 0.000,B 0.000,C 90.000,E1 312.933} C_DIS
LIN {X -0.071,Y -241.593,Z 1607.724,A 0.000,B 0.000,C 90.000,E1 310.297} C_DIS
LIN {X -0.130,Y -249.387,Z 1607.714,A 0.000,B 0.000,C 90.000,E1 308.463} C_DIS
LIN {X 0.148,Y -258.146,Z 1607.703,A 0.000,B 0.000,C 90.000,E1 306.583} C_DIS
LIN {X 0.052,Y -267.819,Z 1607.693,A 0.000,B 0.000,C 90.000,E1 304.818} C_DIS
LIN {X -0.109,Y -280.701,Z 1607.682,A 0.000,B 0.000,C 90.000,E1 302.752} C_DIS
LIN {X 0.063,Y -302.045,Z 1607.665,A 0.000,B 0.000,C 90.000,E1 299.667} C_DIS
LIN {X -0.050,Y -316.994,Z 1607.654,A 0.000,B 0.000,C 90.000,E1 297.719} C_DIS
LIN {X 0.018,Y -329.382,Z 1607.645,A 0.000,B 0.000,C 90.000,E1 296.104} C_DIS
LIN {X 0.148,Y -341.493,Z 1607.636,A 0.000,B 0.000,C 90.000,E1 294.515} C_DIS
LIN {X 0.118,Y -360.795,Z 1607.623,A 0.000,B 0.000,C 90.000,E1 292.078} C_DIS
LIN {X -0.008,Y -372.923,Z 1607.615,A 0.000,B 0.000,C 90.000,E1 290.610} C_DIS
LIN {X -0.185,Y -379.972,Z 1607.610,A 0.000,B 0.000,C 90.000,E1 289.758} C_DIS
LIN {X 0.059,Y -386.449,Z 1607.605,A 0.000,B 0.000,C 90.000,E1 288.852} C_DIS
LIN {X 0.006,Y -392.466,Z 1607.600,A 0.000,B 0.000,C 90.000,E1 288.000} C_DIS
LIN {X -0.003,Y -397.963,Z 1607.595,A 0.000,B 0.000,C 90.000,E1 287.149} C_DIS
LIN {X 0.121,Y -401.266,Z 1607.592,A 0.000,B 0.000,C 90.000,E1 286.567} C_DIS
LIN {X 0.086,Y -405.527,Z 1607.588,A 0.000,B 0.000,C 90.000,E1 285.733} C_DIS
LIN {X 0.084,Y -408.845,Z 1607.583,A 0.000,B 0.000,C 90.000,E1 284.898} C_DIS
LIN {X 0.002,Y -410.590,Z 1607.580,A 0.000,B 0.000,C 90.000,E1 284.356} C_DIS
LIN {X -0.178,Y -411.904,Z 1607.577,A 0.000,B 0.000,C 90.000,E1 283.828} C_DIS
LIN {X 0.054,Y -412.816,Z 1607.574,A 0.000,B 0.000,C 90.000,E1 283.244} C_DIS
LIN {X -0.014,Y -413.267,Z 1607.571,A 0.000,B 0.000,C 90.000,E1 282.703} C_DIS
LIN {X 0.233,Y -413.230,Z 1607.568,A 0.000,B 0.000,C 90.000,E1 282.119} C_DIS
LIN {X 0.079,Y -412.668,Z 1607.564,A 0.000,B 0.000,C 90.000,E1 281.591} C_DIS
LIN {X -0.155,Y -411.591,Z 1607.561,A 0.000,B 0.000,C 90.000,E1 281.074} C_DIS
LIN {X 0.092,Y -409.940,Z 1607.558,A 0.000,B 0.000,C 90.000,E1 280.489} C_DIS
LIN {X -0.070,Y -407.674,Z 1607.555,A 0.000,B 0.000,C 90.000,E1 279.962} C_DIS
LIN {X 0.148,Y -404.733,Z 1607.552,A 0.000,B 0.000,C 90.000,E1 279.378} C_DIS
LIN {X -0.113,Y -401.073,Z 1607.549,A 0.000,B 0.000,C 90.000,E1 278.859} C_DIS
LIN {X 0.065,Y -396.773,Z 1607.546,A 0.000,B 0.000,C 90.000,E1 278.276} C_DIS
LIN {X 0.159,Y -391.881,Z 1607.543,A 0.000,B 0.000,C 90.000,E1 277.701} C_DIS
LIN {X -0.157,Y -386.277,Z 1607.540,A 0.000,B 0.000,C 90.000,E1 277.182} C_DIS
LIN {X -0.147,Y -380.584,Z 1607.537,A 0.000,B 0.000,C 90.000,E1 276.663} C_DIS
LIN {X 0.037,Y -374.553,Z 1607.534,A 0.000,B 0.000,C 90.000,E1 276.144} C_DIS
LIN {X 0.122,Y -368.394,Z 1607.532,A 0.000,B 0.000,C 90.000,E1 275.682} C_DIS
LIN {X 0.077,Y -362.099,Z 1607.529,A 0.000,B 0.000,C 90.000,E1 275.277} C_DIS
LIN {X 0.177,Y -352.403,Z 1607.526,A 0.000,B 0.000,C 90.000,E1 274.702} C_DIS
LIN {X -0.059,Y -342.631,Z 1607.524,A 0.000,B 0.000,C 90.000,E1 274.245} C_DIS
LIN {X 0.028,Y -332.840,Z 1607.521,A 0.000,B 0.000,C 90.000,E1 273.784} C_DIS
LIN {X -0.004,Y -322.803,Z 1607.519,A 0.000,B 0.000,C 90.000,E1 273.383} C_DIS
LIN {X -0.029,Y -313.068,Z 1607.517,A 0.000,B 0.000,C 90.000,E1 273.037} C_DIS
LIN {X 0.118,Y -302.892,Z 1607.515,A 0.000,B 0.000,C 90.000,E1 272.694} C_DIS
LIN {X -0.092,Y -291.558,Z 1607.514,A 0.000,B 0.000,C 90.000,E1 272.465} C_DIS
LIN {X 0.038,Y -283.516,Z 1607.513,A 0.000,B 0.000,C 90.000,E1 272.293} C_DIS
LIN {X 0.001,Y -269.215,Z 1607.512,A 0.000,B 0.000,C 90.000,E1 272.121} C_DIS
LIN {X 0.105,Y -254.216,Z 1607.511,A 0.000,B 0.000,C 90.000,E1 271.949} C_DIS
LIN {X -0.083,Y -228.644,Z 1607.510,A 0.000,B 0.000,C 90.000,E1 271.835} C_DIS
LIN {X 0.105,Y -222.592,Z 1607.510,A 0.000,B 0.000,C 90.000,E1 271.776} C_DIS
LIN {X 0.050,Y -181.297,Z 1607.510,A 0.000,B 0.000,C 90.000,E1 271.776} C_DIS
LIN {X 0.015,Y -181.569,Z 1607.500,A 0.000,B 0.000,C 90.000,E1 270.057} C_DIS
LIN {X 0.002,Y -180.864,Z 1607.472,A 0.000,B 0.000,C 90.000,E1 265.008} C_DIS
LIN {X 0.056,Y -178.978,Z 1607.444,A 0.000,B 0.000,C 90.000,E1 259.926} C_DIS
LIN {X 0.066,Y -177.944,Z 1607.435,A 0.000,B 0.000,C 90.000,E1 258.229} C_DIS
LIN {X 0.080,Y -175.584,Z 1607.411,A 0.000,B 0.000,C 90.000,E1 253.976} C_DIS
LIN {X -0.075,Y -172.310,Z 1607.387,A 0.000,B 0.000,C 90.000,E1 249.752} C_DIS
LIN {X 0.064,Y -171.789,Z 1607.383,A 0.000,B 0.000,C 90.000,E1 248.847} C_DIS
LIN {X -0.059,Y -169.456,Z 1607.368,A 0.000,B 0.000,C 90.000,E1 246.305} C_DIS
LIN {X -0.002,Y -166.786,Z 1607.349,A 0.000,B 0.000,C 90.000,E1 242.820} C_DIS
LIN {X -0.007,Y -162.766,Z 1607.325,A 0.000,B 0.000,C 90.000,E1 238.456} C_DIS
LIN {X -0.032,Y -161.455,Z 1607.315,A 0.000,B 0.000,C 90.000,E1 236.707} C_DIS
LIN {X 0.010,Y -157.450,Z 1607.290,A 0.000,B 0.000,C 90.000,E1 232.271} C_DIS
LIN {X -0.056,Y -155.459,Z 1607.276,A 0.000,B 0.000,C 90.000,E1 229.622} C_DIS
LIN {X -0.015,Y -151.774,Z 1607.251,A 0.000,B 0.000,C 90.000,E1 225.121} C_DIS
LIN {X 0.002,Y -149.979,Z 1607.236,A 0.000,B 0.000,C 90.000,E1 222.405} C_DIS
LIN {X 0.014,Y -146.814,Z 1607.210,A 0.000,B 0.000,C 90.000,E1 217.855} C_DIS
LIN {X 0.030,Y -145.391,Z 1607.195,A 0.000,B 0.000,C 90.000,E1 215.105} C_DIS
LIN {X -0.053,Y -142.828,Z 1607.170,A 0.000,B 0.000,C 90.000,E1 210.541} C_DIS
LIN {X 0.004,Y -141.440,Z 1607.149,A 0.000,B 0.000,C 90.000,E1 206.821} C_DIS
LIN {X 0.048,Y -139.368,Z 1607.113,A 0.000,B 0.000,C 90.000,E1 200.301} C_DIS
LIN {X 0.034,Y -138.815,Z 1607.097,A 0.000,B 0.000,C 90.000,E1 197.511} C_DIS
LIN {X -0.051,Y -138.351,Z 1607.056,A 0.000,B 0.000,C 90.000,E1 190.074} C_DIS
LIN {X 0.062,Y -139.537,Z 1607.004,A 0.000,B 0.000,C 90.000,E1 180.688} C_DIS
LIN {X 0.014,Y -141.227,Z 1606.973,A 0.000,B 0.000,C 90.000,E1 175.122} C_DIS
LIN {X -0.027,Y -142.600,Z 1606.958,A 0.000,B 0.000,C 90.000,E1 172.356} C_DIS
LIN {X 0.068,Y -144.905,Z 1606.932,A 0.000,B 0.000,C 90.000,E1 167.701} C_DIS
LIN {X 0.021,Y -147.533,Z 1606.911,A 0.000,B 0.000,C 90.000,E1 164.047} C_DIS
LIN {X -0.048,Y -150.133,Z 1606.891,A 0.000,B 0.000,C 90.000,E1 160.423} C_DIS
LIN {X -0.037,Y -153.497,Z 1606.871,A 0.000,B 0.000,C 90.000,E1 156.794} C_DIS
LIN {X 0.026,Y -157.863,Z 1606.846,A 0.000,B 0.000,C 90.000,E1 152.281} C_DIS
LIN {X -0.018,Y -162.148,Z 1606.826,A 0.000,B 0.000,C 90.000,E1 148.742} C_DIS
LIN {X -0.039,Y -166.353,Z 1606.807,A 0.000,B 0.000,C 90.000,E1 145.229} C_DIS
LIN {X -0.034,Y -171.370,Z 1606.787,A 0.000,B 0.000,C 90.000,E1 141.743} C_DIS
LIN {X -0.108,Y -176.279,Z 1606.768,A 0.000,B 0.000,C 90.000,E1 138.324} C_DIS
LIN {X 0.011,Y -180.563,Z 1606.754,A 0.000,B 0.000,C 90.000,E1 135.729} C_DIS
LIN {X -0.010,Y -185.965,Z 1606.735,A 0.000,B 0.000,C 90.000,E1 132.366} C_DIS
LIN {X 0.045,Y -190.597,Z 1606.721,A 0.000,B 0.000,C 90.000,E1 129.850} C_DIS
LIN {X -0.047,Y -196.347,Z 1606.703,A 0.000,B 0.000,C 90.000,E1 126.583} C_DIS
LIN {X 0.030,Y -201.142,Z 1606.690,A 0.000,B 0.000,C 90.000,E1 124.119} C_DIS
LIN {X -0.068,Y -205.225,Z 1606.677,A 0.000,B 0.000,C 90.000,E1 121.878} C_DIS
LIN {X -0.143,Y -323.575,Z 1606.677,A 0.000,B 0.000,C 90.000,E1 121.878} C_DIS
LIN {X 0.198,Y -324.909,Z 1606.677,A 0.000,B 0.000,C 90.000,E1 121.799} C_DIS
LIN {X -0.053,Y -328.386,Z 1606.676,A 0.000,B 0.000,C 90.000,E1 121.720} C_DIS
LIN {X 0.139,Y -331.655,Z 1606.675,A 0.000,B 0.000,C 90.000,E1 121.465} C_DIS
LIN {X 0.016,Y -335.342,Z 1606.673,A 0.000,B 0.000,C 90.000,E1 121.082} C_DIS
LIN {X -0.048,Y -337.232,Z 1606.671,A 0.000,B 0.000,C 90.000,E1 120.797} C_DIS
LIN {X 0.179,Y -338.711,Z 1606.669,A 0.000,B 0.000,C 90.000,E1 120.463} C_DIS
LIN {X -0.098,Y -351.926,Z 1606.652,A 0.000,B 0.000,C 90.000,E1 117.436} C_DIS
LIN {X -0.034,Y -365.315,Z 1606.637,A 0.000,B 0.000,C 90.000,E1 114.719} C_DIS
LIN {X -0.073,Y -380.274,Z 1606.623,A 0.000,B 0.000,C 90.000,E1 112.078} C_DIS
LIN {X 0.070,Y -394.987,Z 1606.610,A 0.000,B 0.000,C 90.000,E1 109.758} C_DIS
LIN {X 0.079,Y -411.141,Z 1606.597,A 0.000,B 0.000,C 90.000,E1 107.511} C_DIS
LIN {X 0.122,Y -428.847,Z 1606.585,A 0.000,B 0.000,C 90.000,E1 105.315} C_DIS
LIN {X 0.243,Y -448.163,Z 1606.573,A 0.000,B 0.000,C 90.000,E1 103.175} C_DIS
LIN {X -0.099,Y -468.297,Z 1606.562,A 0.000,B 0.000,C 90.000,E1 101.243} C_DIS
LIN {X -0.082,Y -491.562,Z 1606.551,A 0.000,B 0.000,C 90.000,E1 99.208} C_DIS
LIN {X 0.222,Y -496.681,Z 1606.549,A 0.000,B 0.000,C 90.000,E1 98.746} C_DIS
LIN {X -0.060,Y -498.588,Z 1606.548,A 0.000,B 0.000,C 90.000,E1 98.568} C_DIS
LIN {X -0.214,Y -500.257,Z 1606.546,A 0.000,B 0.000,C 90.000,E1 98.341} C_DIS
LIN {X 0.203,Y -501.505,Z 1606.545,A 0.000,B 0.000,C 90.000,E1 98.049} C_DIS
LIN {X -0.008,Y -503.018,Z 1606.542,A 0.000,B 0.000,C 90.000,E1 97.587} C_DIS
LIN {X -0.211,Y -503.454,Z 1606.539,A 0.000,B 0.000,C 90.000,E1 97.125} C_DIS
LIN {X 0.093,Y -502.889,Z 1606.537,A 0.000,B 0.000,C 90.000,E1 96.606} C_DIS
LIN {X -0.098,Y -501.229,Z 1606.534,A 0.000,B 0.000,C 90.000,E1 96.144} C_DIS
LIN {X -0.170,Y -499.895,Z 1606.533,A 0.000,B 0.000,C 90.000,E1 95.910} C_DIS
LIN {X 0.178,Y -484.924,Z 1606.521,A 0.000,B 0.000,C 90.000,E1 93.669} C_DIS
LIN {X 0.167,Y -474.949,Z 1606.512,A 0.000,B 0.000,C 90.000,E1 92.178} C_DIS
LIN {X 0.186,Y -466.274,Z 1606.505,A 0.000,B 0.000,C 90.000,E1 90.917} C_DIS
LIN {X -0.146,Y -455.441,Z 1606.497,A 0.000,B 0.000,C 90.000,E1 89.427} C_DIS
LIN {X -0.191,Y -444.144,Z 1606.488,A 0.000,B 0.000,C 90.000,E1 87.879} C_DIS
LIN {X -0.148,Y -434.234,Z 1606.481,A 0.000,B 0.000,C 90.000,E1 86.560} C_DIS
LIN {X 0.011,Y -420.102,Z 1606.470,A 0.000,B 0.000,C 90.000,E1 84.666} C_DIS
LIN {X -0.190,Y -400.863,Z 1606.455,A 0.000,B 0.000,C 90.000,E1 81.951} C_DIS
LIN {X -0.030,Y -383.000,Z 1606.439,A 0.000,B 0.000,C 90.000,E1 79.106} C_DIS
LIN {X 0.194,Y -367.839,Z 1606.425,A 0.000,B 0.000,C 90.000,E1 76.464} C_DIS
LIN {X 0.183,Y -356.428,Z 1606.413,A 0.000,B 0.000,C 90.000,E1 74.393} C_DIS
LIN {X 0.063,Y -342.245,Z 1606.398,A 0.000,B 0.000,C 90.000,E1 71.692} C_DIS
LIN {X 0.121,Y -330.011,Z 1606.385,A 0.000,B 0.000,C 90.000,E1 69.209} C_DIS
LIN {X 0.032,Y -314.299,Z 1606.365,A 0.000,B 0.000,C 90.000,E1 65.741} C_DIS
LIN {X 0.144,Y -303.921,Z 1606.351,A 0.000,B 0.000,C 90.000,E1 63.127} C_DIS
LIN {X 0.009,Y -294.879,Z 1606.338,A 0.000,B 0.000,C 90.000,E1 60.845} C_DIS
LIN {X -0.155,Y -286.701,Z 1606.327,A 0.000,B 0.000,C 90.000,E1 58.869} C_DIS
LIN {X 0.099,Y -279.516,Z 1606.318,A 0.000,B 0.000,C 90.000,E1 57.120} C_DIS
LIN {X 0.155,Y -272.084,Z 1606.308,A 0.000,B 0.000,C 90.000,E1 55.388} C_DIS
LIN {X -0.092,Y -260.156,Z 1606.292,A 0.000,B 0.000,C 90.000,E1 52.637} C_DIS
LIN {X 0.024,Y -247.511,Z 1606.274,A 0.000,B 0.000,C 90.000,E1 49.380} C_DIS
LIN {X -0.049,Y -237.401,Z 1606.258,A 0.000,B 0.000,C 90.000,E1 46.458} C_DIS
LIN {X 0.054,Y -227.053,Z 1606.239,A 0.000,B 0.000,C 90.000,E1 43.056} C_DIS
LIN {X 0.006,Y -218.649,Z 1606.222,A 0.000,B 0.000,C 90.000,E1 40.011} C_DIS
LIN {X 0.125,Y -211.002,Z 1606.205,A 0.000,B 0.000,C 90.000,E1 36.870} C_DIS
LIN {X 0.136,Y -204.106,Z 1606.188,A 0.000,B 0.000,C 90.000,E1 33.706} C_DIS
LIN {X -0.012,Y -198.020,Z 1606.170,A 0.000,B 0.000,C 90.000,E1 30.541} C_DIS
LIN {X 0.107,Y -192.646,Z 1606.152,A 0.000,B 0.000,C 90.000,E1 27.257} C_DIS
LIN {X -0.007,Y -187.984,Z 1606.133,A 0.000,B 0.000,C 90.000,E1 24.003} C_DIS
LIN {X 0.103,Y -183.127,Z 1606.110,A 0.000,B 0.000,C 90.000,E1 19.812} C_DIS
LIN {X -0.061,Y -179.053,Z 1606.087,A 0.000,B 0.000,C 90.000,E1 15.662} C_DIS
LIN {X 0.017,Y -175.181,Z 1606.059,A 0.000,B 0.000,C 90.000,E1 10.546} C_DIS
LIN {X 0.085,Y -172.220,Z 1606.025,A 0.000,B 0.000,C 90.000,E1 4.531} C_DIS
LIN {X -0.031,Y -170.745,Z 1605.997,A 0.000,B 0.000,C 90.000,E1 359.542} C_DIS
LIN {X 0.070,Y -171.937,Z 1605.935,A 0.000,B 0.000,C 90.000,E1 348.285} C_DIS
LIN {X 0.031,Y -174.646,Z 1605.906,A 0.000,B 0.000,C 90.000,E1 343.142} C_DIS
LIN {X -0.059,Y -178.328,Z 1605.883,A 0.000,B 0.000,C 90.000,E1 338.901} C_DIS
LIN {X 0.028,Y -182.176,Z 1605.864,A 0.000,B 0.000,C 90.000,E1 335.485} C_DIS
LIN {X -0.056,Y -186.787,Z 1605.845,A 0.000,B 0.000,C 90.000,E1 332.153} C_DIS
LIN {X 0.079,Y -192.219,Z 1605.827,A 0.000,B 0.000,C 90.000,E1 328.791} C_DIS
LIN {X 0.064,Y -198.466,Z 1605.808,A 0.000,B 0.000,C 90.000,E1 325.515} C_DIS
LIN {X 0.101,Y -205.429,Z 1605.791,A 0.000,B 0.000,C 90.000,E1 322.271} C_DIS
LIN {X 0.078,Y -213.321,Z 1605.773,A 0.000,B 0.000,C 90.000,E1 319.094} C_DIS
LIN {X 0.075,Y -222.152,Z 1605.755,A 0.000,B 0.000,C 90.000,E1 315.972} C_DIS
LIN {X -0.022,Y -231.923,Z 1605.739,A 0.000,B 0.000,C 90.000,E1 312.933} C_DIS
LIN {X 0.005,Y -241.518,Z 1605.724,A 0.000,B 0.000,C 90.000,E1 310.297} C_DIS
LIN {X -0.053,Y -249.262,Z 1605.714,A 0.000,B 0.000,C 90.000,E1 308.463} C_DIS
LIN {X -0.136,Y -257.982,Z 1605.703,A 0.000,B 0.000,C 90.000,E1 306.664} C_DIS
LIN {X 0.129,Y -267.664,Z 1605.694,A 0.000,B 0.000,C 90.000,E1 304.818} C_DIS
LIN {X -0.030,Y -280.558,Z 1605.682,A 0.000,B 0.000,C 90.000,E1 302.752} C_DIS
LIN {X 0.143,Y -301.862,Z 1605.665,A 0.000,B 0.000,C 90.000,E1 299.667} C_DIS
LIN {X 0.030,Y -316.846,Z 1605.654,A 0.000,B 0.000,C 90.000,E1 297.719} C_DIS
LIN {X 0.100,Y -329.222,Z 1605.645,A 0.000,B 0.000,C 90.000,E1 296.104} C_DIS
LIN {X -0.080,Y -341.363,Z 1605.636,A 0.000,B 0.000,C 90.000,E1 294.567} C_DIS
LIN {X 0.066,Y -360.684,Z 1605.623,A 0.000,B 0.000,C 90.000,E1 292.099} C_DIS
LIN {X 0.076,Y -372.854,Z 1605.615,A 0.000,B 0.000,C 90.000,E1 290.610} C_DIS
LIN {X -0.098,Y -379.911,Z 1605.610,A 0.000,B 0.000,C 90.000,E1 289.758} C_DIS
LIN {X -0.080,Y -388.538,Z 1605.603,A 0.000,B 0.000,C 90.000,E1 288.598} C_DIS
LIN {X -0.126,Y -394.426,Z 1605.599,A 0.000,B 0.000,C 90.000,E1 287.747} C_DIS
LIN {X 0.147,Y -399.717,Z 1605.594,A 0.000,B 0.000,C 90.000,E1 286.858} C_DIS
LIN {X 0.090,Y -404.313,Z 1605.589,A 0.000,B 0.000,C 90.000,E1 286.024} C_DIS
LIN {X -0.016,Y -406.859,Z 1605.586,A 0.000,B 0.000,C 90.000,E1 285.481} C_DIS
LIN {X -0.218,Y -409.034,Z 1605.583,A 0.000,B 0.000,C 90.000,E1 284.954} C_DIS
LIN {X 0.097,Y -410.782,Z 1605.580,A 0.000,B 0.000,C 90.000,E1 284.356} C_DIS
LIN {X -0.081,Y -412.131,Z 1605.577,A 0.000,B 0.000,C 90.000,E1 283.828} C_DIS
LIN {X 0.153,Y -413.078,Z 1605.574,A 0.000,B 0.000,C 90.000,E1 283.244} C_DIS
LIN {X -0.005,Y -413.531,Z 1605.571,A 0.000,B 0.000,C 90.000,E1 282.715} C_DIS
LIN {X -0.070,Y -413.536,Z 1605.568,A 0.000,B 0.000,C 90.000,E1 282.175} C_DIS
LIN {X 0.182,Y -413.012,Z 1605.565,A 0.000,B 0.000,C 90.000,E1 281.591} C_DIS
LIN {X -0.051,Y -411.968,Z 1605.562,A 0.000,B 0.000,C 90.000,E1 281.074} C_DIS
LIN {X -0.205,Y -410.382,Z 1605.558,A 0.000,B 0.000,C 90.000,E1 280.546} C_DIS
LIN {X 0.037,Y -408.157,Z 1605.555,A 0.000,B 0.000,C 90.000,E1 279.962} C_DIS
LIN {X -0.142,Y -405.229,Z 1605.552,A 0.000,B 0.000,C 90.000,E1 279.434} C_DIS
LIN {X -0.002,Y -401.651,Z 1605.549,A 0.000,B 0.000,C 90.000,E1 278.859} C_DIS
LIN {X 0.178,Y -397.366,Z 1605.546,A 0.000,B 0.000,C 90.000,E1 278.276} C_DIS
LIN {X -0.115,Y -392.517,Z 1605.543,A 0.000,B 0.000,C 90.000,E1 277.757} C_DIS
LIN {X -0.041,Y -386.930,Z 1605.540,A 0.000,B 0.000,C 90.000,E1 277.182} C_DIS
LIN {X -0.071,Y -381.146,Z 1605.537,A 0.000,B 0.000,C 90.000,E1 276.663} C_DIS
LIN {X 0.134,Y -375.142,Z 1605.534,A 0.000,B 0.000,C 90.000,E1 276.144} C_DIS
LIN {X -0.155,Y -368.943,Z 1605.532,A 0.000,B 0.000,C 90.000,E1 275.739} C_DIS
LIN {X -0.170,Y -362.684,Z 1605.530,A 0.000,B 0.000,C 90.000,E1 275.334} C_DIS
LIN {X -0.030,Y -353.108,Z 1605.526,A 0.000,B 0.000,C 90.000,E1 274.759} C_DIS
LIN {X 0.108,Y -343.352,Z 1605.524,A 0.000,B 0.000,C 90.000,E1 274.245} C_DIS
LIN {X -0.058,Y -333.974,Z 1605.521,A 0.000,B 0.000,C 90.000,E1 273.841} C_DIS
LIN {X -0.064,Y -324.154,Z 1605.519,A 0.000,B 0.000,C 90.000,E1 273.440} C_DIS
LIN {X -0.136,Y -314.240,Z 1605.517,A 0.000,B 0.000,C 90.000,E1 273.094} C_DIS
LIN {X -0.004,Y -304.141,Z 1605.515,A 0.000,B 0.000,C 90.000,E1 272.751} C_DIS
LIN {X 0.058,Y -293.000,Z 1605.514,A 0.000,B 0.000,C 90.000,E1 272.465} C_DIS
LIN {X -0.117,Y -285.096,Z 1605.513,A 0.000,B 0.000,C 90.000,E1 272.350} C_DIS
LIN {X 0.114,Y -271.179,Z 1605.512,A 0.000,B 0.000,C 90.000,E1 272.121} C_DIS
LIN {X -0.052,Y -256.531,Z 1605.511,A 0.000,B 0.000,C 90.000,E1 272.007} C_DIS
LIN {X 0.089,Y -235.052,Z 1605.510,A 0.000,B 0.000,C 90.000,E1 271.835} C_DIS
LIN {X -0.044,Y -228.239,Z 1605.510,A 0.000,B 0.000,C 90.000,E1 271.835} C_DIS
LIN {X -0.084,Y -220.371,Z 1605.510,A 0.000,B 0.000,C 90.000,E1 271.835} C_DIS
LIN {X 0.083,Y -181.296,Z 1605.510,A 0.000,B 0.000,C 90.000,E1 271.776} C_DIS
LIN {X 0.086,Y -181.571,Z 1605.500,A 0.000,B 0.000,C 90.000,E1 270.057} C_DIS
LIN {X 0.074,Y -180.869,Z 1605.472,A 0.000,B 0.000,C 90.000,E1 265.008} C_DIS
LIN {X -0.049,Y -178.983,Z 1605.444,A 0.000,B 0.000,C 90.000,E1 259.982} C_DIS
LIN {X -0.038,Y -177.959,Z 1605.435,A 0.000,B 0.000,C 90.000,E1 258.285} C_DIS
LIN {X -0.019,Y -175.601,Z 1605.411,A 0.000,B 0.000,C 90.000,E1 254.031} C_DIS
LIN {X -0.006,Y -172.325,Z 1605.387,A 0.000,B 0.000,C 90.000,E1 249.752} C_DIS
LIN {X -0.028,Y -171.802,Z 1605.383,A 0.000,B 0.000,C 90.000,E1 248.901} C_DIS
LIN {X 0.010,Y -169.476,Z 1605.368,A 0.000,B 0.000,C 90.000,E1 246.305} C_DIS
LIN {X -0.083,Y -166.804,Z 1605.349,A 0.000,B 0.000,C 90.000,E1 242.871} C_DIS
LIN {X 0.060,Y -162.784,Z 1605.325,A 0.000,B 0.000,C 90.000,E1 238.456} C_DIS
LIN {X 0.035,Y -161.473,Z 1605.315,A 0.000,B 0.000,C 90.000,E1 236.707} C_DIS
LIN {X 0.077,Y -157.468,Z 1605.291,A 0.000,B 0.000,C 90.000,E1 232.271} C_DIS
LIN {X 0.008,Y -155.482,Z 1605.276,A 0.000,B 0.000,C 90.000,E1 229.622} C_DIS
LIN {X -0.059,Y -151.791,Z 1605.251,A 0.000,B 0.000,C 90.000,E1 225.162} C_DIS
LIN {X -0.046,Y -149.999,Z 1605.236,A 0.000,B 0.000,C 90.000,E1 222.447} C_DIS
LIN {X -0.014,Y -146.828,Z 1605.210,A 0.000,B 0.000,C 90.000,E1 217.890} C_DIS
LIN {X -0.027,Y -145.408,Z 1605.195,A 0.000,B 0.000,C 90.000,E1 215.152} C_DIS
LIN {X 0.009,Y -142.839,Z 1605.170,A 0.000,B 0.000,C 90.000,E1 210.541} C_DIS
LIN {X -0.061,Y -141.452,Z 1605.149,A 0.000,B 0.000,C 90.000,E1 206.873} C_DIS
LIN {X -0.021,Y -139.373,Z 1605.113,A 0.000,B 0.000,C 90.000,E1 200.355} C_DIS
LIN {X -0.079,Y -138.822,Z 1605.098,A 0.000,B 0.000,C 90.000,E1 197.583} C_DIS
LIN {X 0.010,Y -138.353,Z 1605.056,A 0.000,B 0.000,C 90.000,E1 190.074} C_DIS
LIN {X -0.018,Y -139.534,Z 1605.004,A 0.000,B 0.000,C 90.000,E1 180.745} C_DIS
LIN {X -0.066,Y -141.216,Z 1604.973,A 0.000,B 0.000,C 90.000,E1 175.179} C_DIS
LIN {X 0.035,Y -142.590,Z 1604.958,A 0.000,B 0.000,C 90.000,E1 172.356} C_DIS
LIN {X -0.012,Y -144.890,Z 1604.932,A 0.000,B 0.000,C 90.000,E1 167.757} C_DIS
LIN {X -0.058,Y -147.517,Z 1604.911,A 0.000,B 0.000,C 90.000,E1 164.102} C_DIS
LIN {X 0.016,Y -150.113,Z 1604.891,A 0.000,B 0.000,C 90.000,E1 160.423} C_DIS
LIN {X 0.028,Y -153.472,Z 1604.871,A 0.000,B 0.000,C 90.000,E1 156.794} C_DIS
LIN {X 0.019,Y -157.836,Z 1604.846,A 0.000,B 0.000,C 90.000,E1 152.308} C_DIS
LIN {X 0.049,Y -162.120,Z 1604.826,A 0.000,B 0.000,C 90.000,E1 148.742} C_DIS
LIN {X -0.065,Y -166.323,Z 1604.807,A 0.000,B 0.000,C 90.000,E1 145.261} C_DIS
LIN {X 0.036,Y -171.340,Z 1604.787,A 0.000,B 0.000,C 90.000,E1 141.743} C_DIS
LIN {X -0.037,Y -176.242,Z 1604.768,A 0.000,B 0.000,C 90.000,E1 138.324} C_DIS
LIN {X 0.082,Y -180.523,Z 1604.754,A 0.000,B 0.000,C 90.000,E1 135.729} C_DIS
LIN {X 0.062,Y -185.926,Z 1604.735,A 0.000,B 0.000,C 90.000,E1 132.366} C_DIS
LIN {X -0.002,Y -190.555,Z 1604.722,A 0.000,B 0.000,C 90.000,E1 129.886} C_DIS
LIN {X 0.028,Y -196.306,Z 1604.703,A 0.000,B 0.000,C 90.000,E1 126.583} C_DIS
LIN {X 0.107,Y -201.105,Z 1604.690,A 0.000,B 0.000,C 90.000,E1 124.119} C_DIS
LIN {X 0.078,Y -205.147,Z 1604.677,A 0.000,B 0.000,C 90.000,E1 121.878} C_DIS
LIN {X 0.087,Y -323.300,Z 1604.677,A 0.000,B 0.000,C 90.000,E1 121.878} C_DIS
LIN {X 0.017,Y -324.344,Z 1604.677,A 0.000,B 0.000,C 90.000,E1 121.878} C_DIS
LIN {X 0.070,Y -328.552,Z 1604.676,A 0.000,B 0.000,C 90.000,E1 121.720} C_DIS
LIN {X -0.016,Y -331.679,Z 1604.675,A 0.000,B 0.000,C 90.000,E1 121.514} C_DIS
LIN {X 0.057,Y -335.395,Z 1604.673,A 0.000,B 0.000,C 90.000,E1 121.082} C_DIS
LIN {X -0.041,Y -337.264,Z 1604.671,A 0.000,B 0.000,C 90.000,E1 120.797} C_DIS
LIN {X 0.149,Y -338.727,Z 1604.669,A 0.000,B 0.000,C 90.000,E1 120.463} C_DIS
